LIN {X 123.176,Y 42.359,Z 55.000,A 180.000,B 0.000,C 180.000} C_DIS
LIN {X 122.928,Y 42.550,Z 55.000,A 180.000,B 0.000,C 180.000} C_DIS
LIN {X 122.818,Y 42.627,Z 55.000,A 180.000,B 0.000,C 180.000} C_DIS
LIN {X 122.639,Y 42.749,Z 55.000,A 180.000,B 0.000,C 180.000} C_DIS
LIN {X 122.461,Y 42.865,Z 55.000,A 180.000,B 0.000,C 180.000} C_DIS
LIN {X 122.282,Y 42.971,Z 55.000,A 180.000,B 0.000,C 180.000} C_DIS
LIN {X 122.103,Y 43.076,Z 55.000,A 180.000,B 0.000,C 180.000} C_DIS
LIN {X 121.731,Y 43.266,Z 55.000,A 180.000,B 0.000,C 180.000} C_DIS
LIN {X 121.567,Y 43.340,Z 55.000,A 180.000,B 0.000,C 180.000} C_DIS
LIN {X 121.325,Y 43.444,Z 55.000,A 180.000,B 0.000,C 180.000} C_DIS
LIN {X 121.209,Y 43.491,Z 55.000,A 180.000,B 0.000,C 180.000} C_DIS
LIN {X 120.841,Y 43.623,Z 55.000,A 180.000,B 0.000,C 180.000} C_DIS
LIN {X 120.673,Y 43.674,Z 55.000,A 180.000,B 0.000,C 180.000} C_DIS
LIN {X 120.494,Y 43.726,Z 55.000,A 180.000,B 0.000,C 180.000} C_DIS
LIN {X 120.315,Y 43.774,Z 55.000,A 180.000,B 0.000,C 180.000} C_DIS
LIN {X 119.958,Y 43.854,Z 55.000,A 180.000,B 0.000,C 180.000} C_DIS
LIN {X 119.779,Y 43.886,Z 55.000,A 180.000,B 0.000,C 180.000} C_DIS
LIN {X 119.632,Y 43.909,Z 55.000,A 180.000,B 0.000,C 180.000} C_DIS
; Link Move Starts
LIN {X 119.319,Y 43.951,Z 55.000,A 180.000,B 0.000,C 180.000} C_DIS
LIN {X 119.006,Y 43.981,Z 54.999,A 180.000,B 0.000,C 180.000} C_DIS
LIN {X 118.691,Y 43.993,Z 54.998,A 180.000,B 0.000,C 180.000} C_DIS
LIN {X 118.376,Y 43.995,Z 54.996,A 180.000,B 0.000,C 180.000} C_DIS
LIN {X 118.061,Y 43.985,Z 54.994,A 180.000,B 0.000,C 180.000} C_DIS
LIN {X 117.748,Y 43.957,Z 54.991,A 180.000,B 0.000,C 180.000} C_DIS
LIN {X 117.435,Y 43.920,Z 54.988,A 180.000,B 0.000,C 180.000} C_DIS
LIN {X 117.124,Y 43.871,Z 54.985,A 180.000,B 0.000,C 180.000} C_DIS
LIN {X 116.816,Y 43.804,Z 54.981,A 180.000,B 0.000,C 180.000} C_DIS
LIN {X 116.510,Y 43.727,Z 54.977,A 180.000,B 0.000,C 180.000} C_DIS
LIN {X 116.208,Y 43.639,Z 54.972,A 180.000,B 0.000,C 180.000} C_DIS
LIN {X 116.059,Y 43.587,Z 54.969,A 180.000,B 0.000,C 180.000} C_DIS
LIN {X 115.911,Y 43.534,Z 54.967,A 180.000,B 0.000,C 180.000} C_DIS
LIN {X 115.763,Y 43.481,Z 54.964,A 180.000,B 0.000,C 180.000} C_DIS
LIN {X 115.618,Y 43.419,Z 54.961,A 180.000,B 0.000,C 180.000} C_DIS
LIN {X 115.473,Y 43.357,Z 54.959,A 180.000,B 0.000,C 180.000} C_DIS
LIN {X 115.329,Y 43.294,Z 54.956,A 180.000,B 0.000,C 180.000} C_DIS
LIN {X 115.188,Y 43.224,Z 54.952,A 180.000,B 0.000,C 180.000} C_DIS
LIN {X 115.047,Y 43.153,Z 54.949,A 180.000,B 0.000,C 180.000} C_DIS
LIN {X 114.907,Y 43.081,Z 54.946,A 180.000,B 0.000,C 180.000} C_DIS
LIN {X 114.771,Y 43.002,Z 54.943,A 180.000,B 0.000,C 180.000} C_DIS
LIN {X 114.635,Y 42.922,Z 54.939,A 180.000,B 0.000,C 180.000} C_DIS
LIN {X 114.500,Y 42.842,Z 54.936,A 180.000,B 0.000,C 180.000} C_DIS
LIN {X 114.369,Y 42.754,Z 54.932,A 180.000,B 0.000,C 180.000} C_DIS
LIN {X 114.238,Y 42.666,Z 54.928,A 180.000,B 0.000,C 180.000} C_DIS
LIN {X 114.108,Y 42.577,Z 54.925,A 180.000,B 0.000,C 180.000} C_DIS
LIN {X 113.983,Y 42.482,Z 54.921,A 180.000,B 0.000,C 180.000} C_DIS
LIN {X 113.858,Y 42.385,Z 54.917,A 180.000,B 0.000,C 180.000} C_DIS
LIN {X 113.734,Y 42.289,Z 54.913,A 180.000,B 0.000,C 180.000} C_DIS
LIN {X 113.615,Y 42.185,Z 54.909,A 180.000,B 0.000,C 180.000} C_DIS
LIN {X 113.497,Y 42.081,Z 54.905,A 180.000,B 0.000,C 180.000} C_DIS
LIN {X 113.379,Y 41.977,Z 54.900,A 180.000,B 0.000,C 180.000} C_DIS
LIN {X 113.267,Y 41.866,Z 54.896,A 180.000,B 0.000,C 180.000} C_DIS
LIN {X 113.155,Y 41.755,Z 54.892,A 180.000,B 0.000,C 180.000} C_DIS
LIN {X 113.044,Y 41.644,Z 54.887,A 180.000,B 0.000,C 180.000} C_DIS
LIN {X 112.939,Y 41.526,Z 54.883,A 180.000,B 0.000,C 180.000} C_DIS
LIN {X 112.835,Y 41.408,Z 54.878,A 180.000,B 0.000,C 180.000} C_DIS
LIN {X 112.731,Y 41.290,Z 54.873,A 180.000,B 0.000,C 180.000} C_DIS
LIN {X 112.634,Y 41.166,Z 54.869,A 180.000,B 0.000,C 180.000} C_DIS
LIN {X 112.537,Y 41.041,Z 54.864,A 180.000,B 0.000,C 180.000} C_DIS
LIN {X 112.441,Y 40.917,Z 54.859,A 180.000,B 0.000,C 180.000} C_DIS
LIN {X 112.351,Y 40.787,Z 54.854,A 180.000,B 0.000,C 180.000} C_DIS
LIN {X 112.307,Y 40.722,Z 54.851,A 180.000,B 0.000,C 180.000} C_DIS
LIN {X 112.263,Y 40.657,Z 54.849,A 180.000,B 0.000,C 180.000} C_DIS
LIN {X 112.219,Y 40.592,Z 54.846,A 180.000,B 0.000,C 180.000} C_DIS
LIN {X 112.174,Y 40.526,Z 54.844,A 180.000,B 0.000,C 180.000} C_DIS
LIN {X 112.134,Y 40.459,Z 54.841,A 180.000,B 0.000,C 180.000} C_DIS
LIN {X 112.094,Y 40.391,Z 54.839,A 180.000,B 0.000,C 180.000} C_DIS
LIN {X 112.053,Y 40.323,Z 54.836,A 180.000,B 0.000,C 180.000} C_DIS
LIN {X 111.973,Y 40.188,Z 54.831,A 180.000,B 0.000,C 180.000} C_DIS
LIN {X 111.933,Y 40.120,Z 54.828,A 180.000,B 0.000,C 180.000} C_DIS
LIN {X 111.897,Y 40.050,Z 54.825,A 180.000,B 0.000,C 180.000} C_DIS
LIN {X 111.825,Y 39.910,Z 54.820,A 180.000,B 0.000,C 180.000} C_DIS
LIN {X 111.754,Y 39.769,Z 54.815,A 180.000,B 0.000,C 180.000} C_DIS
LIN {X 111.718,Y 39.699,Z 54.812,A 180.000,B 0.000,C 180.000} C_DIS
LIN {X 111.687,Y 39.627,Z 54.809,A 180.000,B 0.000,C 180.000} C_DIS
LIN {X 111.655,Y 39.555,Z 54.806,A 180.000,B 0.000,C 180.000} C_DIS
LIN {X 111.593,Y 39.410,Z 54.801,A 180.000,B 0.000,C 180.000} C_DIS
LIN {X 111.530,Y 39.266,Z 54.795,A 180.000,B 0.000,C 180.000} C_DIS
LIN {X 111.503,Y 39.192,Z 54.793,A 180.000,B 0.000,C 180.000} C_DIS
LIN {X 111.450,Y 39.044,Z 54.787,A 180.000,B 0.000,C 180.000} C_DIS
LIN {X 111.423,Y 38.969,Z 54.785,A 180.000,B 0.000,C 180.000} C_DIS
LIN {X 111.370,Y 38.821,Z 54.779,A 180.000,B 0.000,C 180.000} C_DIS
LIN {X 111.347,Y 38.746,Z 54.776,A 180.000,B 0.000,C 180.000} C_DIS
LIN {X 111.326,Y 38.670,Z 54.774,A 180.000,B 0.000,C 180.000} C_DIS
LIN {X 111.282,Y 38.519,Z 54.768,A 180.000,B 0.000,C 180.000} C_DIS
LIN {X 111.238,Y 38.368,Z 54.763,A 180.000,B 0.000,C 180.000} C_DIS
LIN {X 111.220,Y 38.291,Z 54.760,A 180.000,B 0.000,C 180.000} C_DIS
LIN {X 111.186,Y 38.137,Z 54.754,A 180.000,B 0.000,C 180.000} C_DIS
LIN {X 111.169,Y 38.060,Z 54.752,A 180.000,B 0.000,C 180.000} C_DIS
LIN {X 111.134,Y 37.906,Z 54.746,A 180.000,B 0.000,C 180.000} C_DIS
LIN {X 111.122,Y 37.829,Z 54.743,A 180.000,B 0.000,C 180.000} C_DIS
LIN {X 111.110,Y 37.751,Z 54.741,A 180.000,B 0.000,C 180.000} C_DIS
LIN {X 111.085,Y 37.595,Z 54.735,A 180.000,B 0.000,C 180.000} C_DIS
LIN {X 111.060,Y 37.440,Z 54.730,A 180.000,B 0.000,C 180.000} C_DIS
LIN {X 111.046,Y 37.283,Z 54.724,A 180.000,B 0.000,C 180.000} C_DIS
LIN {X 111.023,Y 37.048,Z 54.716,A 180.000,B 0.000,C 180.000} C_DIS
LIN {X 111.016,Y 36.969,Z 54.713,A 180.000,B 0.000,C 180.000} C_DIS
LIN {X 111.004,Y 36.576,Z 54.699,A 180.000,B 0.000,C 180.000} C_DIS
LIN {X 111.001,Y 36.497,Z 54.697,A 180.000,B 0.000,C 180.000} C_DIS
LIN {X 111.006,Y 36.340,Z 54.691,A 180.000,B 0.000,C 180.000} C_DIS
LIN {X 111.014,Y 36.103,Z 54.683,A 180.000,B 0.000,C 180.000} C_DIS
LIN {X 111.016,Y 36.025,Z 54.680,A 180.000,B 0.000,C 180.000} C_DIS
LIN {X 111.054,Y 35.633,Z 54.666,A 180.000,B 0.000,C 180.000} C_DIS
LIN {X 111.061,Y 35.554,Z 54.664,A 180.000,B 0.000,C 180.000} C_DIS
LIN {X 111.098,Y 35.321,Z 54.655,A 180.000,B 0.000,C 180.000} C_DIS
LIN {X 111.123,Y 35.165,Z 54.650,A 180.000,B 0.000,C 180.000} C_DIS
LIN {X 111.136,Y 35.088,Z 54.647,A 180.000,B 0.000,C 180.000} C_DIS
LIN {X 111.222,Y 34.703,Z 54.633,A 180.000,B 0.000,C 180.000} C_DIS
LIN {X 111.239,Y 34.627,Z 54.631,A 180.000,B 0.000,C 180.000} C_DIS
LIN {X 111.305,Y 34.400,Z 54.622,A 180.000,B 0.000,C 180.000} C_DIS
LIN {X 111.349,Y 34.248,Z 54.617,A 180.000,B 0.000,C 180.000} C_DIS
LIN {X 111.372,Y 34.173,Z 54.614,A 180.000,B 0.000,C 180.000} C_DIS
LIN {X 111.505,Y 33.802,Z 54.600,A 180.000,B 0.000,C 180.000} C_DIS
LIN {X 111.533,Y 33.729,Z 54.598,A 180.000,B 0.000,C 180.000} C_DIS
LIN {X 111.626,Y 33.512,Z 54.589,A 180.000,B 0.000,C 180.000} C_DIS
LIN {X 111.689,Y 33.367,Z 54.584,A 180.000,B 0.000,C 180.000} C_DIS
LIN {X 111.721,Y 33.295,Z 54.581,A 180.000,B 0.000,C 180.000} C_DIS
LIN {X 111.900,Y 32.944,Z 54.567,A 180.000,B 0.000,C 180.000} C_DIS
LIN {X 111.936,Y 32.875,Z 54.565,A 180.000,B 0.000,C 180.000} C_DIS
LIN {X 112.137,Y 32.536,Z 54.551,A 180.000,B 0.000,C 180.000} C_DIS
LIN {X 112.178,Y 32.468,Z 54.548,A 180.000,B 0.000,C 180.000} C_DIS
LIN {X 112.399,Y 32.143,Z 54.534,A 180.000,B 0.000,C 180.000} C_DIS
LIN {X 112.444,Y 32.078,Z 54.532,A 180.000,B 0.000,C 180.000} C_DIS
LIN {X 112.686,Y 31.767,Z 54.518,A 180.000,B 0.000,C 180.000} C_DIS
LIN {X 112.735,Y 31.706,Z 54.515,A 180.000,B 0.000,C 180.000} C_DIS
LIN {X 112.995,Y 31.410,Z 54.501,A 180.000,B 0.000,C 180.000} C_DIS
LIN {X 113.048,Y 31.352,Z 54.499,A 180.000,B 0.000,C 180.000} C_DIS
LIN {X 113.327,Y 31.074,Z 54.485,A 180.000,B 0.000,C 180.000} C_DIS
LIN {X 113.383,Y 31.019,Z 54.482,A 180.000,B 0.000,C 180.000} C_DIS
LIN {X 113.679,Y 30.759,Z 54.468,A 180.000,B 0.000,C 180.000} C_DIS
LIN {X 113.739,Y 30.708,Z 54.466,A 180.000,B 0.000,C 180.000} C_DIS
LIN {X 114.050,Y 30.466,Z 54.452,A 180.000,B 0.000,C 180.000} C_DIS
LIN {X 114.113,Y 30.419,Z 54.449,A 180.000,B 0.000,C 180.000} C_DIS
LIN {X 114.439,Y 30.198,Z 54.435,A 180.000,B 0.000,C 180.000} C_DIS
LIN {X 114.505,Y 30.155,Z 54.433,A 180.000,B 0.000,C 180.000} C_DIS
LIN {X 114.844,Y 29.955,Z 54.419,A 180.000,B 0.000,C 180.000} C_DIS
LIN {X 114.913,Y 29.916,Z 54.416,A 180.000,B 0.000,C 180.000} C_DIS
LIN {X 115.263,Y 29.737,Z 54.402,A 180.000,B 0.000,C 180.000} C_DIS
LIN {X 115.334,Y 29.703,Z 54.400,A 180.000,B 0.000,C 180.000} C_DIS
LIN {X 115.551,Y 29.609,Z 54.391,A 180.000,B 0.000,C 180.000} C_DIS
LIN {X 115.696,Y 29.547,Z 54.386,A 180.000,B 0.000,C 180.000} C_DIS
LIN {X 115.769,Y 29.517,Z 54.383,A 180.000,B 0.000,C 180.000} C_DIS
LIN {X 116.139,Y 29.384,Z 54.369,A 180.000,B 0.000,C 180.000} C_DIS
LIN {X 116.214,Y 29.359,Z 54.367,A 180.000,B 0.000,C 180.000} C_DIS
LIN {X 116.441,Y 29.293,Z 54.358,A 180.000,B 0.000,C 180.000} C_DIS
LIN {X 116.592,Y 29.249,Z 54.353,A 180.000,B 0.000,C 180.000} C_DIS
LIN {X 116.668,Y 29.229,Z 54.350,A 180.000,B 0.000,C 180.000} C_DIS
LIN {X 117.053,Y 29.144,Z 54.336,A 180.000,B 0.000,C 180.000} C_DIS
LIN {X 117.130,Y 29.129,Z 54.334,A 180.000,B 0.000,C 180.000} C_DIS
LIN {X 117.285,Y 29.104,Z 54.328,A 180.000,B 0.000,C 180.000} C_DIS
LIN {X 117.519,Y 29.067,Z 54.320,A 180.000,B 0.000,C 180.000} C_DIS
LIN {X 117.597,Y 29.057,Z 54.317,A 180.000,B 0.000,C 180.000} C_DIS
LIN {X 117.989,Y 29.020,Z 54.303,A 180.000,B 0.000,C 180.000} C_DIS
LIN {X 118.068,Y 29.015,Z 54.301,A 180.000,B 0.000,C 180.000} C_DIS
LIN {X 118.225,Y 29.010,Z 54.295,A 180.000,B 0.000,C 180.000} C_DIS
LIN {X 118.461,Y 29.002,Z 54.287,A 180.000,B 0.000,C 180.000} C_DIS
LIN {X 118.540,Y 29.002,Z 54.284,A 180.000,B 0.000,C 180.000} C_DIS
LIN {X 118.776,Y 29.010,Z 54.276,A 180.000,B 0.000,C 180.000} C_DIS
LIN {X 118.933,Y 29.015,Z 54.270,A 180.000,B 0.000,C 180.000} C_DIS
LIN {X 119.012,Y 29.020,Z 54.268,A 180.000,B 0.000,C 180.000} C_DIS
LIN {X 119.169,Y 29.035,Z 54.262,A 180.000,B 0.000,C 180.000} C_DIS
LIN {X 119.404,Y 29.057,Z 54.254,A 180.000,B 0.000,C 180.000} C_DIS
LIN {X 119.482,Y 29.067,Z 54.251,A 180.000,B 0.000,C 180.000} C_DIS
LIN {X 119.716,Y 29.104,Z 54.243,A 180.000,B 0.000,C 180.000} C_DIS
LIN {X 119.871,Y 29.129,Z 54.237,A 180.000,B 0.000,C 180.000} C_DIS
LIN {X 119.948,Y 29.144,Z 54.235,A 180.000,B 0.000,C 180.000} C_DIS
LIN {X 120.102,Y 29.178,Z 54.229,A 180.000,B 0.000,C 180.000} C_DIS
LIN {X 120.333,Y 29.230,Z 54.221,A 180.000,B 0.000,C 180.000} C_DIS
LIN {X 120.409,Y 29.250,Z 54.218,A 180.000,B 0.000,C 180.000} C_DIS
LIN {X 120.636,Y 29.316,Z 54.210,A 180.000,B 0.000,C 180.000} C_DIS
LIN {X 120.787,Y 29.359,Z 54.204,A 180.000,B 0.000,C 180.000} C_DIS
LIN {X 120.862,Y 29.384,Z 54.202,A 180.000,B 0.000,C 180.000} C_DIS
LIN {X 121.010,Y 29.438,Z 54.196,A 180.000,B 0.000,C 180.000} C_DIS
LIN {X 121.158,Y 29.491,Z 54.191,A 180.000,B 0.000,C 180.000} C_DIS
LIN {X 121.232,Y 29.518,Z 54.188,A 180.000,B 0.000,C 180.000} C_DIS
LIN {X 121.305,Y 29.547,Z 54.185,A 180.000,B 0.000,C 180.000} C_DIS
LIN {X 121.450,Y 29.610,Z 54.180,A 180.000,B 0.000,C 180.000} C_DIS
LIN {X 121.594,Y 29.672,Z 54.174,A 180.000,B 0.000,C 180.000} C_DIS
LIN {X 121.667,Y 29.704,Z 54.172,A 180.000,B 0.000,C 180.000} C_DIS
LIN {X 121.738,Y 29.738,Z 54.169,A 180.000,B 0.000,C 180.000} C_DIS
LIN {X 121.878,Y 29.809,Z 54.164,A 180.000,B 0.000,C 180.000} C_DIS
LIN {X 121.948,Y 29.845,Z 54.161,A 180.000,B 0.000,C 180.000} C_DIS
LIN {X 122.018,Y 29.881,Z 54.159,A 180.000,B 0.000,C 180.000} C_DIS
LIN {X 122.088,Y 29.917,Z 54.156,A 180.000,B 0.000,C 180.000} C_DIS
LIN {X 122.157,Y 29.955,Z 54.154,A 180.000,B 0.000,C 180.000} C_DIS
LIN {X 122.225,Y 29.995,Z 54.151,A 180.000,B 0.000,C 180.000} C_DIS
LIN {X 122.293,Y 30.035,Z 54.149,A 180.000,B 0.000,C 180.000} C_DIS
LIN {X 122.428,Y 30.115,Z 54.144,A 180.000,B 0.000,C 180.000} C_DIS
LIN {X 122.562,Y 30.198,Z 54.139,A 180.000,B 0.000,C 180.000} C_DIS
LIN {X 122.692,Y 30.287,Z 54.134,A 180.000,B 0.000,C 180.000} C_DIS
LIN {X 122.823,Y 30.376,Z 54.129,A 180.000,B 0.000,C 180.000} C_DIS
LIN {X 122.951,Y 30.467,Z 54.124,A 180.000,B 0.000,C 180.000} C_DIS
LIN {X 123.075,Y 30.563,Z 54.120,A 180.000,B 0.000,C 180.000} C_DIS
LIN {X 123.200,Y 30.660,Z 54.115,A 180.000,B 0.000,C 180.000} C_DIS
LIN {X 123.322,Y 30.759,Z 54.111,A 180.000,B 0.000,C 180.000} C_DIS
LIN {X 123.440,Y 30.863,Z 54.106,A 180.000,B 0.000,C 180.000} C_DIS
LIN {X 123.558,Y 30.968,Z 54.102,A 180.000,B 0.000,C 180.000} C_DIS
LIN {X 123.674,Y 31.074,Z 54.097,A 180.000,B 0.000,C 180.000} C_DIS
LIN {X 123.785,Y 31.186,Z 54.093,A 180.000,B 0.000,C 180.000} C_DIS
LIN {X 123.897,Y 31.297,Z 54.089,A 180.000,B 0.000,C 180.000} C_DIS
LIN {X 124.006,Y 31.411,Z 54.085,A 180.000,B 0.000,C 180.000} C_DIS
LIN {X 124.110,Y 31.529,Z 54.081,A 180.000,B 0.000,C 180.000} C_DIS
LIN {X 124.214,Y 31.647,Z 54.077,A 180.000,B 0.000,C 180.000} C_DIS
LIN {X 124.315,Y 31.768,Z 54.073,A 180.000,B 0.000,C 180.000} C_DIS
LIN {X 124.412,Y 31.893,Z 54.070,A 180.000,B 0.000,C 180.000} C_DIS
LIN {X 124.508,Y 32.017,Z 54.066,A 180.000,B 0.000,C 180.000} C_DIS
LIN {X 124.602,Y 32.144,Z 54.062,A 180.000,B 0.000,C 180.000} C_DIS
LIN {X 124.690,Y 32.274,Z 54.059,A 180.000,B 0.000,C 180.000} C_DIS
LIN {X 124.779,Y 32.404,Z 54.056,A 180.000,B 0.000,C 180.000} C_DIS
LIN {X 124.864,Y 32.537,Z 54.052,A 180.000,B 0.000,C 180.000} C_DIS
LIN {X 124.944,Y 32.672,Z 54.049,A 180.000,B 0.000,C 180.000} C_DIS
LIN {X 125.024,Y 32.808,Z 54.046,A 180.000,B 0.000,C 180.000} C_DIS
LIN {X 125.101,Y 32.945,Z 54.043,A 180.000,B 0.000,C 180.000} C_DIS
LIN {X 125.172,Y 33.086,Z 54.040,A 180.000,B 0.000,C 180.000} C_DIS
LIN {X 125.244,Y 33.226,Z 54.037,A 180.000,B 0.000,C 180.000} C_DIS
LIN {X 125.312,Y 33.368,Z 54.034,A 180.000,B 0.000,C 180.000} C_DIS
LIN {X 125.374,Y 33.513,Z 54.032,A 180.000,B 0.000,C 180.000} C_DIS
LIN {X 125.437,Y 33.657,Z 54.029,A 180.000,B 0.000,C 180.000} C_DIS
LIN {X 125.495,Y 33.804,Z 54.027,A 180.000,B 0.000,C 180.000} C_DIS
LIN {X 125.602,Y 34.100,Z 54.022,A 180.000,B 0.000,C 180.000} C_DIS
LIN {X 125.695,Y 34.401,Z 54.018,A 180.000,B 0.000,C 180.000} C_DIS
LIN {X 125.779,Y 34.705,Z 54.014,A 180.000,B 0.000,C 180.000} C_DIS
LIN {X 125.847,Y 35.012,Z 54.011,A 180.000,B 0.000,C 180.000} C_DIS
LIN {X 125.902,Y 35.322,Z 54.008,A 180.000,B 0.000,C 180.000} C_DIS
LIN {X 125.947,Y 35.634,Z 54.005,A 180.000,B 0.000,C 180.000} C_DIS
LIN {X 125.976,Y 35.947,Z 54.003,A 180.000,B 0.000,C 180.000} C_DIS
LIN {X 125.991,Y 36.262,Z 54.002,A 180.000,B 0.000,C 180.000} C_DIS
LIN {X 125.996,Y 36.577,Z 54.001,A 180.000,B 0.000,C 180.000} C_DIS
LIN {X 125.986,Y 36.892,Z 54.000,A 180.000,B 0.000,C 180.000} C_DIS
LIN {X 125.970,Y 37.123,Z 54.000,A 180.000,B 0.000,C 180.000} C_DIS
; Cutting Move Starts
LIN {X 125.947,Y 37.366,Z 54.000,A 180.000,B 0.000,C 180.000} C_DIS
LIN {X 125.923,Y 37.545,Z 54.000,A 180.000,B 0.000,C 180.000} C_DIS
LIN {X 125.866,Y 37.902,Z 54.000,A 180.000,B 0.000,C 180.000} C_DIS
LIN {X 125.857,Y 37.944,Z 54.000,A 180.000,B 0.000,C 180.000} C_DIS
LIN {X 125.787,Y 38.260,Z 54.000,A 180.000,B 0.000,C 180.000} C_DIS
LIN {X 125.742,Y 38.439,Z 54.000,A 180.000,B 0.000,C 180.000} C_DIS
LIN {X 125.638,Y 38.796,Z 54.000,A 180.000,B 0.000,C 180.000} C_DIS
LIN {X 125.575,Y 38.975,Z 54.000,A 180.000,B 0.000,C 180.000} C_DIS
LIN {X 125.500,Y 39.184,Z 54.000,A 180.000,B 0.000,C 180.000} C_DIS
LIN {X 125.441,Y 39.333,Z 54.000,A 180.000,B 0.000,C 180.000} C_DIS
LIN {X 125.286,Y 39.690,Z 54.000,A 180.000,B 0.000,C 180.000} C_DIS
LIN {X 125.195,Y 39.869,Z 54.000,A 180.000,B 0.000,C 180.000} C_DIS
LIN {X 125.104,Y 40.048,Z 54.000,A 180.000,B 0.000,C 180.000} C_DIS
LIN {X 125.004,Y 40.226,Z 54.000,A 180.000,B 0.000,C 180.000} C_DIS
LIN {X 124.898,Y 40.405,Z 54.000,A 180.000,B 0.000,C 180.000} C_DIS
LIN {X 124.787,Y 40.584,Z 54.000,A 180.000,B 0.000,C 180.000} C_DIS
LIN {X 124.606,Y 40.850,Z 54.000,A 180.000,B 0.000,C 180.000} C_DIS
LIN {X 124.540,Y 40.942,Z 54.000,A 180.000,B 0.000,C 180.000} C_DIS
LIN {X 124.402,Y 41.120,Z 54.000,A 180.000,B 0.000,C 180.000} C_DIS
LIN {X 124.261,Y 41.299,Z 54.000,A 180.000,B 0.000,C 180.000} C_DIS
LIN {X 124.070,Y 41.516,Z 54.000,A 180.000,B 0.000,C 180.000} C_DIS
LIN {X 123.943,Y 41.657,Z 54.000,A 180.000,B 0.000,C 180.000} C_DIS
LIN {X 123.712,Y 41.888,Z 54.000,A 180.000,B 0.000,C 180.000} C_DIS
LIN {X 123.579,Y 42.014,Z 54.000,A 180.000,B 0.000,C 180.000} C_DIS
LIN {X 123.354,Y 42.212,Z 54.000,A 180.000,B 0.000,C 180.000} C_DIS
LIN {X 123.176,Y 42.359,Z 54.000,A 180.000,B 0.000,C 180.000} C_DIS
LIN {X 122.928,Y 42.550,Z 54.000,A 180.000,B 0.000,C 180.000} C_DIS
LIN {X 122.818,Y 42.627,Z 54.000,A 180.000,B 0.000,C 180.000} C_DIS
LIN {X 122.639,Y 42.749,Z 54.000,A 180.000,B 0.000,C 180.000} C_DIS
LIN {X 122.461,Y 42.865,Z 54.000,A 180.000,B 0.000,C 180.000} C_DIS
LIN {X 122.282,Y 42.971,Z 54.000,A 180.000,B 0.000,C 180.000} C_DIS
LIN {X 122.103,Y 43.076,Z 54.000,A 180.000,B 0.000,C 180.000} C_DIS
LIN {X 121.731,Y 43.266,Z 54.000,A 180.000,B 0.000,C 180.000} C_DIS
LIN {X 121.567,Y 43.340,Z 54.000,A 180.000,B 0.000,C 180.000} C_DIS
LIN {X 121.325,Y 43.444,Z 54.000,A 180.000,B 0.000,C 180.000} C_DIS
LIN {X 121.209,Y 43.491,Z 54.000,A 180.000,B 0.000,C 180.000} C_DIS
LIN {X 120.841,Y 43.623,Z 54.000,A 180.000,B 0.000,C 180.000} C_DIS
LIN {X 120.673,Y 43.674,Z 54.000,A 180.000,B 0.000,C 180.000} C_DIS
LIN {X 120.494,Y 43.726,Z 54.000,A 180.000,B 0.000,C 180.000} C_DIS
LIN {X 120.315,Y 43.774,Z 54.000,A 180.000,B 0.000,C 180.000} C_DIS
LIN {X 119.958,Y 43.854,Z 54.000,A 180.000,B 0.000,C 180.000} C_DIS
LIN {X 119.779,Y 43.886,Z 54.000,A 180.000,B 0.000,C 180.000} C_DIS
LIN {X 119.632,Y 43.909,Z 54.000,A 180.000,B 0.000,C 180.000} C_DIS
LIN {X 119.600,Y 43.914,Z 54.000,A 180.000,B 0.000,C 180.000} C_DIS
LIN {X 119.422,Y 43.941,Z 54.000,A 180.000,B 0.000,C 180.000} C_DIS
LIN {X 119.006,Y 43.981,Z 54.000,A 180.000,B 0.000,C 180.000} C_DIS
LIN {X 118.885,Y 43.987,Z 54.000,A 180.000,B 0.000,C 180.000} C_DIS
LIN {X 118.528,Y 43.998,Z 54.000,A 180.000,B 0.000,C 180.000} C_DIS
LIN {X 118.349,Y 43.994,Z 54.000,A 180.000,B 0.000,C 180.000} C_DIS
LIN {X 118.170,Y 43.988,Z 54.000,A 180.000,B 0.000,C 180.000} C_DIS
LIN {X 117.994,Y 43.981,Z 54.000,A 180.000,B 0.000,C 180.000} C_DIS
LIN {X 117.634,Y 43.947,Z 54.000,A 180.000,B 0.000,C 180.000} C_DIS
LIN {X 117.455,Y 43.923,Z 54.000,A 180.000,B 0.000,C 180.000} C_DIS
LIN {X 117.098,Y 43.866,Z 54.000,A 180.000,B 0.000,C 180.000} C_DIS
LIN {X 116.919,Y 43.827,Z 54.000,A 180.000,B 0.000,C 180.000} C_DIS
LIN {X 116.740,Y 43.787,Z 54.000,A 180.000,B 0.000,C 180.000} C_DIS
LIN {X 116.561,Y 43.742,Z 54.000,A 180.000,B 0.000,C 180.000} C_DIS
LIN {X 116.204,Y 43.638,Z 54.000,A 180.000,B 0.000,C 180.000} C_DIS
LIN {X 116.159,Y 43.623,Z 54.000,A 180.000,B 0.000,C 180.000} C_DIS
LIN {X 115.846,Y 43.511,Z 54.000,A 180.000,B 0.000,C 180.000} C_DIS
LIN {X 115.675,Y 43.444,Z 54.000,A 180.000,B 0.000,C 180.000} C_DIS
LIN {X 115.310,Y 43.286,Z 54.000,A 180.000,B 0.000,C 180.000} C_DIS
LIN {X 115.269,Y 43.266,Z 54.000,A 180.000,B 0.000,C 180.000} C_DIS
LIN {X 114.918,Y 43.087,Z 54.000,A 180.000,B 0.000,C 180.000} C_DIS
LIN {X 114.774,Y 43.004,Z 54.000,A 180.000,B 0.000,C 180.000} C_DIS
LIN {X 114.595,Y 42.898,Z 54.000,A 180.000,B 0.000,C 180.000} C_DIS
LIN {X 114.416,Y 42.787,Z 54.000,A 180.000,B 0.000,C 180.000} C_DIS
LIN {X 114.237,Y 42.665,Z 54.000,A 180.000,B 0.000,C 180.000} C_DIS
LIN {X 114.072,Y 42.550,Z 54.000,A 180.000,B 0.000,C 180.000} C_DIS
LIN {X 113.841,Y 42.372,Z 54.000,A 180.000,B 0.000,C 180.000} C_DIS
LIN {X 113.701,Y 42.261,Z 54.000,A 180.000,B 0.000,C 180.000} C_DIS
LIN {X 113.421,Y 42.014,Z 54.000,A 180.000,B 0.000,C 180.000} C_DIS
LIN {X 113.343,Y 41.943,Z 54.000,A 180.000,B 0.000,C 180.000} C_DIS
LIN {X 113.057,Y 41.657,Z 54.000,A 180.000,B 0.000,C 180.000} C_DIS
LIN {X 112.986,Y 41.579,Z 54.000,A 180.000,B 0.000,C 180.000} C_DIS
LIN {X 112.739,Y 41.299,Z 54.000,A 180.000,B 0.000,C 180.000} C_DIS
LIN {X 112.628,Y 41.159,Z 54.000,A 180.000,B 0.000,C 180.000} C_DIS
LIN {X 112.450,Y 40.928,Z 54.000,A 180.000,B 0.000,C 180.000} C_DIS
LIN {X 112.335,Y 40.763,Z 54.000,A 180.000,B 0.000,C 180.000} C_DIS
LIN {X 112.213,Y 40.584,Z 54.000,A 180.000,B 0.000,C 180.000} C_DIS
LIN {X 112.102,Y 40.405,Z 54.000,A 180.000,B 0.000,C 180.000} C_DIS
LIN {X 111.996,Y 40.226,Z 54.000,A 180.000,B 0.000,C 180.000} C_DIS
LIN {X 111.913,Y 40.082,Z 54.000,A 180.000,B 0.000,C 180.000} C_DIS
LIN {X 111.734,Y 39.731,Z 54.000,A 180.000,B 0.000,C 180.000} C_DIS
LIN {X 111.714,Y 39.690,Z 54.000,A 180.000,B 0.000,C 180.000} C_DIS
LIN {X 111.556,Y 39.325,Z 54.000,A 180.000,B 0.000,C 180.000} C_DIS
LIN {X 111.489,Y 39.154,Z 54.000,A 180.000,B 0.000,C 180.000} C_DIS
LIN {X 111.377,Y 38.841,Z 54.000,A 180.000,B 0.000,C 180.000} C_DIS
LIN {X 111.362,Y 38.796,Z 54.000,A 180.000,B 0.000,C 180.000} C_DIS
LIN {X 111.258,Y 38.439,Z 54.000,A 180.000,B 0.000,C 180.000} C_DIS
LIN {X 111.213,Y 38.260,Z 54.000,A 180.000,B 0.000,C 180.000} C_DIS
LIN {X 111.173,Y 38.081,Z 54.000,A 180.000,B 0.000,C 180.000} C_DIS
LIN {X 111.134,Y 37.902,Z 54.000,A 180.000,B 0.000,C 180.000} C_DIS
LIN {X 111.077,Y 37.545,Z 54.000,A 180.000,B 0.000,C 180.000} C_DIS
LIN {X 111.053,Y 37.366,Z 54.000,A 180.000,B 0.000,C 180.000} C_DIS
LIN {X 111.019,Y 37.006,Z 54.000,A 180.000,B 0.000,C 180.000} C_DIS
LIN {X 111.012,Y 36.830,Z 54.000,A 180.000,B 0.000,C 180.000} C_DIS
LIN {X 111.006,Y 36.651,Z 54.000,A 180.000,B 0.000,C 180.000} C_DIS
LIN {X 111.002,Y 36.472,Z 54.000,A 180.000,B 0.000,C 180.000} C_DIS
LIN {X 111.013,Y 36.115,Z 54.000,A 180.000,B 0.000,C 180.000} C_DIS
LIN {X 111.019,Y 35.994,Z 54.000,A 180.000,B 0.000,C 180.000} C_DIS
LIN {X 111.059,Y 35.578,Z 54.000,A 180.000,B 0.000,C 180.000} C_DIS
LIN {X 111.086,Y 35.400,Z 54.000,A 180.000,B 0.000,C 180.000} C_DIS
LIN {X 111.114,Y 35.221,Z 54.000,A 180.000,B 0.000,C 180.000} C_DIS
LIN {X 111.146,Y 35.042,Z 54.000,A 180.000,B 0.000,C 180.000} C_DIS
LIN {X 111.226,Y 34.685,Z 54.000,A 180.000,B 0.000,C 180.000} C_DIS
LIN {X 111.274,Y 34.506,Z 54.000,A 180.000,B 0.000,C 180.000} C_DIS
LIN {X 111.326,Y 34.327,Z 54.000,A 180.000,B 0.000,C 180.000} C_DIS
LIN {X 111.377,Y 34.159,Z 54.000,A 180.000,B 0.000,C 180.000} C_DIS
LIN {X 111.509,Y 33.791,Z 54.000,A 180.000,B 0.000,C 180.000} C_DIS
LIN {X 111.556,Y 33.675,Z 54.000,A 180.000,B 0.000,C 180.000} C_DIS
LIN {X 111.660,Y 33.433,Z 54.000,A 180.000,B 0.000,C 180.000} C_DIS
LIN {X 111.734,Y 33.269,Z 54.000,A 180.000,B 0.000,C 180.000} C_DIS
LIN {X 111.924,Y 32.897,Z 54.000,A 180.000,B 0.000,C 180.000} C_DIS
LIN {X 112.029,Y 32.718,Z 54.000,A 180.000,B 0.000,C 180.000} C_DIS
LIN {X 112.135,Y 32.539,Z 54.000,A 180.000,B 0.000,C 180.000} C_DIS
LIN {X 112.251,Y 32.361,Z 54.000,A 180.000,B 0.000,C 180.000} C_DIS
LIN {X 112.373,Y 32.182,Z 54.000,A 180.000,B 0.000,C 180.000} C_DIS
LIN {X 112.450,Y 32.072,Z 54.000,A 180.000,B 0.000,C 180.000} C_DIS
LIN {X 112.641,Y 31.824,Z 54.000,A 180.000,B 0.000,C 180.000} C_DIS
LIN {X 112.788,Y 31.646,Z 54.000,A 180.000,B 0.000,C 180.000} C_DIS
LIN {X 112.986,Y 31.421,Z 54.000,A 180.000,B 0.000,C 180.000} C_DIS
LIN {X 113.112,Y 31.288,Z 54.000,A 180.000,B 0.000,C 180.000} C_DIS
LIN {X 113.343,Y 31.057,Z 54.000,A 180.000,B 0.000,C 180.000} C_DIS
LIN {X 113.484,Y 30.930,Z 54.000,A 180.000,B 0.000,C 180.000} C_DIS
LIN {X 113.701,Y 30.739,Z 54.000,A 180.000,B 0.000,C 180.000} C_DIS
LIN {X 113.880,Y 30.598,Z 54.000,A 180.000,B 0.000,C 180.000} C_DIS
LIN {X 114.058,Y 30.460,Z 54.000,A 180.000,B 0.000,C 180.000} C_DIS
LIN {X 114.150,Y 30.394,Z 54.000,A 180.000,B 0.000,C 180.000} C_DIS
LIN {X 114.416,Y 30.213,Z 54.000,A 180.000,B 0.000,C 180.000} C_DIS
LIN {X 114.595,Y 30.102,Z 54.000,A 180.000,B 0.000,C 180.000} C_DIS
LIN {X 114.774,Y 29.996,Z 54.000,A 180.000,B 0.000,C 180.000} C_DIS
LIN {X 114.952,Y 29.896,Z 54.000,A 180.000,B 0.000,C 180.000} C_DIS
LIN {X 115.131,Y 29.805,Z 54.000,A 180.000,B 0.000,C 180.000} C_DIS
LIN {X 115.310,Y 29.714,Z 54.000,A 180.000,B 0.000,C 180.000} C_DIS
LIN {X 115.667,Y 29.559,Z 54.000,A 180.000,B 0.000,C 180.000} C_DIS
LIN {X 115.816,Y 29.500,Z 54.000,A 180.000,B 0.000,C 180.000} C_DIS
LIN {X 116.025,Y 29.425,Z 54.000,A 180.000,B 0.000,C 180.000} C_DIS
LIN {X 116.204,Y 29.362,Z 54.000,A 180.000,B 0.000,C 180.000} C_DIS
LIN {X 116.561,Y 29.258,Z 54.000,A 180.000,B 0.000,C 180.000} C_DIS
LIN {X 116.740,Y 29.213,Z 54.000,A 180.000,B 0.000,C 180.000} C_DIS
LIN {X 117.056,Y 29.143,Z 54.000,A 180.000,B 0.000,C 180.000} C_DIS
LIN {X 117.098,Y 29.134,Z 54.000,A 180.000,B 0.000,C 180.000} C_DIS
LIN {X 117.455,Y 29.077,Z 54.000,A 180.000,B 0.000,C 180.000} C_DIS
LIN {X 117.634,Y 29.053,Z 54.000,A 180.000,B 0.000,C 180.000} C_DIS
LIN {X 117.991,Y 29.020,Z 54.000,A 180.000,B 0.000,C 180.000} C_DIS
LIN {X 118.170,Y 29.012,Z 54.000,A 180.000,B 0.000,C 180.000} C_DIS
LIN {X 118.349,Y 29.006,Z 54.000,A 180.000,B 0.000,C 180.000} C_DIS
LIN {X 118.528,Y 29.002,Z 54.000,A 180.000,B 0.000,C 180.000} C_DIS
LIN {X 118.885,Y 29.013,Z 54.000,A 180.000,B 0.000,C 180.000} C_DIS
LIN {X 119.064,Y 29.025,Z 54.000,A 180.000,B 0.000,C 180.000} C_DIS
LIN {X 119.422,Y 29.059,Z 54.000,A 180.000,B 0.000,C 180.000} C_DIS
LIN {X 119.600,Y 29.086,Z 54.000,A 180.000,B 0.000,C 180.000} C_DIS
LIN {X 119.779,Y 29.114,Z 54.000,A 180.000,B 0.000,C 180.000} C_DIS
LIN {X 119.944,Y 29.143,Z 54.000,A 180.000,B 0.000,C 180.000} C_DIS
LIN {X 120.315,Y 29.226,Z 54.000,A 180.000,B 0.000,C 180.000} C_DIS
LIN {X 120.494,Y 29.274,Z 54.000,A 180.000,B 0.000,C 180.000} C_DIS
LIN {X 120.673,Y 29.326,Z 54.000,A 180.000,B 0.000,C 180.000} C_DIS
LIN {X 120.852,Y 29.381,Z 54.000,A 180.000,B 0.000,C 180.000} C_DIS
LIN {X 121.209,Y 29.509,Z 54.000,A 180.000,B 0.000,C 180.000} C_DIS
LIN {X 121.388,Y 29.583,Z 54.000,A 180.000,B 0.000,C 180.000} C_DIS
LIN {X 121.610,Y 29.679,Z 54.000,A 180.000,B 0.000,C 180.000} C_DIS
LIN {X 121.746,Y 29.742,Z 54.000,A 180.000,B 0.000,C 180.000} C_DIS
LIN {X 122.103,Y 29.924,Z 54.000,A 180.000,B 0.000,C 180.000} C_DIS
LIN {X 122.282,Y 30.029,Z 54.000,A 180.000,B 0.000,C 180.000} C_DIS
LIN {X 122.461,Y 30.135,Z 54.000,A 180.000,B 0.000,C 180.000} C_DIS
LIN {X 122.587,Y 30.215,Z 54.000,A 180.000,B 0.000,C 180.000} C_DIS
LIN {X 122.850,Y 30.394,Z 54.000,A 180.000,B 0.000,C 180.000} C_DIS
LIN {X 122.997,Y 30.503,Z 54.000,A 180.000,B 0.000,C 180.000} C_DIS
LIN {X 123.176,Y 30.641,Z 54.000,A 180.000,B 0.000,C 180.000} C_DIS
LIN {X 123.313,Y 30.752,Z 54.000,A 180.000,B 0.000,C 180.000} C_DIS
LIN {X 123.533,Y 30.945,Z 54.000,A 180.000,B 0.000,C 180.000} C_DIS
LIN {X 123.709,Y 31.109,Z 54.000,A 180.000,B 0.000,C 180.000} C_DIS
LIN {X 123.891,Y 31.291,Z 54.000,A 180.000,B 0.000,C 180.000} C_DIS
LIN {X 124.055,Y 31.467,Z 54.000,A 180.000,B 0.000,C 180.000} C_DIS
LIN {X 124.248,Y 31.687,Z 54.000,A 180.000,B 0.000,C 180.000} C_DIS
LIN {X 124.359,Y 31.824,Z 54.000,A 180.000,B 0.000,C 180.000} C_DIS
LIN {X 124.497,Y 32.003,Z 54.000,A 180.000,B 0.000,C 180.000} C_DIS
LIN {X 124.606,Y 32.150,Z 54.000,A 180.000,B 0.000,C 180.000} C_DIS
LIN {X 124.785,Y 32.413,Z 54.000,A 180.000,B 0.000,C 180.000} C_DIS
LIN {X 124.865,Y 32.539,Z 54.000,A 180.000,B 0.000,C 180.000} C_DIS
LIN {X 124.971,Y 32.718,Z 54.000,A 180.000,B 0.000,C 180.000} C_DIS
LIN {X 125.076,Y 32.897,Z 54.000,A 180.000,B 0.000,C 180.000} C_DIS
LIN {X 125.258,Y 33.254,Z 54.000,A 180.000,B 0.000,C 180.000} C_DIS
LIN {X 125.321,Y 33.390,Z 54.000,A 180.000,B 0.000,C 180.000} C_DIS
LIN {X 125.417,Y 33.612,Z 54.000,A 180.000,B 0.000,C 180.000} C_DIS
LIN {X 125.491,Y 33.791,Z 54.000,A 180.000,B 0.000,C 180.000} C_DIS
LIN {X 125.619,Y 34.148,Z 54.000,A 180.000,B 0.000,C 180.000} C_DIS
LIN {X 125.674,Y 34.327,Z 54.000,A 180.000,B 0.000,C 180.000} C_DIS
LIN {X 125.726,Y 34.506,Z 54.000,A 180.000,B 0.000,C 180.000} C_DIS
LIN {X 125.774,Y 34.685,Z 54.000,A 180.000,B 0.000,C 180.000} C_DIS
LIN {X 125.857,Y 35.056,Z 54.000,A 180.000,B 0.000,C 180.000} C_DIS
LIN {X 125.886,Y 35.221,Z 54.000,A 180.000,B 0.000,C 180.000} C_DIS
LIN {X 125.914,Y 35.400,Z 54.000,A 180.000,B 0.000,C 180.000} C_DIS
LIN {X 125.941,Y 35.578,Z 54.000,A 180.000,B 0.000,C 180.000} C_DIS
LIN {X 125.975,Y 35.936,Z 54.000,A 180.000,B 0.000,C 180.000} C_DIS
LIN {X 125.987,Y 36.115,Z 54.000,A 180.000,B 0.000,C 180.000} C_DIS
LIN {X 125.998,Y 36.472,Z 54.000,A 180.000,B 0.000,C 180.000} C_DIS
LIN {X 125.994,Y 36.651,Z 54.000,A 180.000,B 0.000,C 180.000} C_DIS
LIN {X 125.988,Y 36.830,Z 54.000,A 180.000,B 0.000,C 180.000} C_DIS
LIN {X 125.980,Y 37.009,Z 54.000,A 180.000,B 0.000,C 180.000} C_DIS
LIN {X 125.970,Y 37.123,Z 54.000,A 180.000,B 0.000,C 180.000} C_DIS
; Link Move Starts
LIN {X 125.940,Y 37.437,Z 54.000,A 180.000,B 0.000,C 180.000} C_DIS
LIN {X 125.891,Y 37.748,Z 53.999,A 180.000,B 0.000,C 180.000} C_DIS
LIN {X 125.832,Y 38.057,Z 53.998,A 180.000,B 0.000,C 180.000} C_DIS
LIN {X 125.763,Y 38.365,Z 53.996,A 180.000,B 0.000,C 180.000} C_DIS
LIN {X 125.675,Y 38.667,Z 53.994,A 180.000,B 0.000,C 180.000} C_DIS
LIN {X 125.578,Y 38.967,Z 53.991,A 180.000,B 0.000,C 180.000} C_DIS
LIN {X 125.471,Y 39.263,Z 53.988,A 180.000,B 0.000,C 180.000} C_DIS
LIN {X 125.346,Y 39.552,Z 53.985,A 180.000,B 0.000,C 180.000} C_DIS
LIN {X 125.212,Y 39.837,Z 53.981,A 180.000,B 0.000,C 180.000} C_DIS
LIN {X 125.068,Y 40.118,Z 53.977,A 180.000,B 0.000,C 180.000} C_DIS
LIN {X 124.908,Y 40.389,Z 53.972,A 180.000,B 0.000,C 180.000} C_DIS
LIN {X 124.827,Y 40.524,Z 53.969,A 180.000,B 0.000,C 180.000} C_DIS
LIN {X 124.739,Y 40.654,Z 53.967,A 180.000,B 0.000,C 180.000} C_DIS
LIN {X 124.650,Y 40.785,Z 53.964,A 180.000,B 0.000,C 180.000} C_DIS
LIN {X 124.561,Y 40.915,Z 53.961,A 180.000,B 0.000,C 180.000} C_DIS
LIN {X 124.465,Y 41.039,Z 53.959,A 180.000,B 0.000,C 180.000} C_DIS
LIN {X 124.368,Y 41.164,Z 53.956,A 180.000,B 0.000,C 180.000} C_DIS
LIN {X 124.271,Y 41.288,Z 53.952,A 180.000,B 0.000,C 180.000} C_DIS
LIN {X 124.167,Y 41.406,Z 53.949,A 180.000,B 0.000,C 180.000} C_DIS
LIN {X 124.063,Y 41.524,Z 53.946,A 180.000,B 0.000,C 180.000} C_DIS
LIN {X 123.958,Y 41.642,Z 53.943,A 180.000,B 0.000,C 180.000} C_DIS
LIN {X 123.847,Y 41.753,Z 53.939,A 180.000,B 0.000,C 180.000} C_DIS
LIN {X 123.735,Y 41.864,Z 53.936,A 180.000,B 0.000,C 180.000} C_DIS
LIN {X 123.623,Y 41.975,Z 53.932,A 180.000,B 0.000,C 180.000} C_DIS
LIN {X 123.505,Y 42.079,Z 53.928,A 180.000,B 0.000,C 180.000} C_DIS
LIN {X 123.387,Y 42.183,Z 53.925,A 180.000,B 0.000,C 180.000} C_DIS
LIN {X 123.268,Y 42.287,Z 53.921,A 180.000,B 0.000,C 180.000} C_DIS
LIN {X 123.144,Y 42.383,Z 53.917,A 180.000,B 0.000,C 180.000} C_DIS
LIN {X 123.019,Y 42.480,Z 53.913,A 180.000,B 0.000,C 180.000} C_DIS
LIN {X 122.894,Y 42.576,Z 53.909,A 180.000,B 0.000,C 180.000} C_DIS
LIN {X 122.764,Y 42.664,Z 53.905,A 180.000,B 0.000,C 180.000} C_DIS
LIN {X 122.634,Y 42.753,Z 53.900,A 180.000,B 0.000,C 180.000} C_DIS
LIN {X 122.503,Y 42.840,Z 53.896,A 180.000,B 0.000,C 180.000} C_DIS
LIN {X 122.367,Y 42.921,Z 53.892,A 180.000,B 0.000,C 180.000} C_DIS
LIN {X 122.232,Y 43.001,Z 53.887,A 180.000,B 0.000,C 180.000} C_DIS
LIN {X 122.095,Y 43.080,Z 53.883,A 180.000,B 0.000,C 180.000} C_DIS
LIN {X 121.955,Y 43.151,Z 53.878,A 180.000,B 0.000,C 180.000} C_DIS
LIN {X 121.815,Y 43.223,Z 53.873,A 180.000,B 0.000,C 180.000} C_DIS
LIN {X 121.674,Y 43.293,Z 53.869,A 180.000,B 0.000,C 180.000} C_DIS
LIN {X 121.529,Y 43.356,Z 53.864,A 180.000,B 0.000,C 180.000} C_DIS
LIN {X 121.385,Y 43.418,Z 53.859,A 180.000,B 0.000,C 180.000} C_DIS
LIN {X 121.240,Y 43.480,Z 53.854,A 180.000,B 0.000,C 180.000} C_DIS
LIN {X 121.166,Y 43.506,Z 53.851,A 180.000,B 0.000,C 180.000} C_DIS
LIN {X 121.091,Y 43.533,Z 53.849,A 180.000,B 0.000,C 180.000} C_DIS
LIN {X 121.017,Y 43.560,Z 53.846,A 180.000,B 0.000,C 180.000} C_DIS
LIN {X 120.943,Y 43.586,Z 53.844,A 180.000,B 0.000,C 180.000} C_DIS
LIN {X 120.869,Y 43.613,Z 53.841,A 180.000,B 0.000,C 180.000} C_DIS
LIN {X 120.795,Y 43.638,Z 53.839,A 180.000,B 0.000,C 180.000} C_DIS
LIN {X 120.719,Y 43.660,Z 53.836,A 180.000,B 0.000,C 180.000} C_DIS
LIN {X 120.568,Y 43.704,Z 53.831,A 180.000,B 0.000,C 180.000} C_DIS
LIN {X 120.416,Y 43.748,Z 53.825,A 180.000,B 0.000,C 180.000} C_DIS
LIN {X 120.340,Y 43.769,Z 53.823,A 180.000,B 0.000,C 180.000} C_DIS
LIN {X 120.187,Y 43.803,Z 53.817,A 180.000,B 0.000,C 180.000} C_DIS
LIN {X 120.033,Y 43.837,Z 53.812,A 180.000,B 0.000,C 180.000} C_DIS
LIN {X 119.956,Y 43.855,Z 53.809,A 180.000,B 0.000,C 180.000} C_DIS
LIN {X 119.879,Y 43.870,Z 53.806,A 180.000,B 0.000,C 180.000} C_DIS
LIN {X 119.723,Y 43.895,Z 53.801,A 180.000,B 0.000,C 180.000} C_DIS
LIN {X 119.490,Y 43.932,Z 53.793,A 180.000,B 0.000,C 180.000} C_DIS
LIN {X 119.412,Y 43.942,Z 53.790,A 180.000,B 0.000,C 180.000} C_DIS
LIN {X 119.177,Y 43.965,Z 53.782,A 180.000,B 0.000,C 180.000} C_DIS
LIN {X 119.020,Y 43.979,Z 53.776,A 180.000,B 0.000,C 180.000} C_DIS
LIN {X 118.941,Y 43.985,Z 53.774,A 180.000,B 0.000,C 180.000} C_DIS
LIN {X 118.784,Y 43.990,Z 53.768,A 180.000,B 0.000,C 180.000} C_DIS
LIN {X 118.548,Y 43.997,Z 53.760,A 180.000,B 0.000,C 180.000} C_DIS
LIN {X 118.469,Y 43.998,Z 53.757,A 180.000,B 0.000,C 180.000} C_DIS
LIN {X 118.233,Y 43.990,Z 53.749,A 180.000,B 0.000,C 180.000} C_DIS
LIN {X 118.075,Y 43.985,Z 53.743,A 180.000,B 0.000,C 180.000} C_DIS
LIN {X 117.997,Y 43.981,Z 53.741,A 180.000,B 0.000,C 180.000} C_DIS
LIN {X 117.840,Y 43.966,Z 53.735,A 180.000,B 0.000,C 180.000} C_DIS
LIN {X 117.605,Y 43.944,Z 53.727,A 180.000,B 0.000,C 180.000} C_DIS
LIN {X 117.527,Y 43.934,Z 53.724,A 180.000,B 0.000,C 180.000} C_DIS
LIN {X 117.138,Y 43.873,Z 53.710,A 180.000,B 0.000,C 180.000} C_DIS
LIN {X 117.060,Y 43.858,Z 53.708,A 180.000,B 0.000,C 180.000} C_DIS
LIN {X 116.907,Y 43.824,Z 53.702,A 180.000,B 0.000,C 180.000} C_DIS
LIN {X 116.676,Y 43.772,Z 53.694,A 180.000,B 0.000,C 180.000} C_DIS
LIN {X 116.600,Y 43.753,Z 53.691,A 180.000,B 0.000,C 180.000} C_DIS
LIN {X 116.222,Y 43.643,Z 53.677,A 180.000,B 0.000,C 180.000} C_DIS
LIN {X 116.147,Y 43.619,Z 53.675,A 180.000,B 0.000,C 180.000} C_DIS
LIN {X 115.999,Y 43.565,Z 53.669,A 180.000,B 0.000,C 180.000} C_DIS
LIN {X 115.776,Y 43.485,Z 53.661,A 180.000,B 0.000,C 180.000} C_DIS
LIN {X 115.703,Y 43.456,Z 53.658,A 180.000,B 0.000,C 180.000} C_DIS
LIN {X 115.342,Y 43.300,Z 53.644,A 180.000,B 0.000,C 180.000} C_DIS
LIN {X 115.270,Y 43.266,Z 53.642,A 180.000,B 0.000,C 180.000} C_DIS
LIN {X 115.060,Y 43.159,Z 53.633,A 180.000,B 0.000,C 180.000} C_DIS
LIN {X 114.920,Y 43.088,Z 53.628,A 180.000,B 0.000,C 180.000} C_DIS
LIN {X 114.851,Y 43.049,Z 53.625,A 180.000,B 0.000,C 180.000} C_DIS
LIN {X 114.512,Y 42.849,Z 53.611,A 180.000,B 0.000,C 180.000} C_DIS
LIN {X 114.445,Y 42.807,Z 53.609,A 180.000,B 0.000,C 180.000} C_DIS
LIN {X 114.250,Y 42.674,Z 53.600,A 180.000,B 0.000,C 180.000} C_DIS
LIN {X 114.120,Y 42.585,Z 53.595,A 180.000,B 0.000,C 180.000} C_DIS
LIN {X 114.056,Y 42.539,Z 53.592,A 180.000,B 0.000,C 180.000} C_DIS
LIN {X 113.745,Y 42.297,Z 53.578,A 180.000,B 0.000,C 180.000} C_DIS
LIN {X 113.685,Y 42.247,Z 53.576,A 180.000,B 0.000,C 180.000} C_DIS
LIN {X 113.389,Y 41.986,Z 53.562,A 180.000,B 0.000,C 180.000} C_DIS
LIN {X 113.332,Y 41.932,Z 53.559,A 180.000,B 0.000,C 180.000} C_DIS
LIN {X 113.054,Y 41.654,Z 53.545,A 180.000,B 0.000,C 180.000} C_DIS
LIN {X 113.001,Y 41.596,Z 53.543,A 180.000,B 0.000,C 180.000} C_DIS
LIN {X 112.740,Y 41.300,Z 53.529,A 180.000,B 0.000,C 180.000} C_DIS
LIN {X 112.691,Y 41.239,Z 53.526,A 180.000,B 0.000,C 180.000} C_DIS
LIN {X 112.449,Y 40.928,Z 53.512,A 180.000,B 0.000,C 180.000} C_DIS
LIN {X 112.404,Y 40.864,Z 53.510,A 180.000,B 0.000,C 180.000} C_DIS
LIN {X 112.182,Y 40.538,Z 53.496,A 180.000,B 0.000,C 180.000} C_DIS
LIN {X 112.141,Y 40.471,Z 53.493,A 180.000,B 0.000,C 180.000} C_DIS
LIN {X 111.940,Y 40.132,Z 53.479,A 180.000,B 0.000,C 180.000} C_DIS
LIN {X 111.903,Y 40.063,Z 53.477,A 180.000,B 0.000,C 180.000} C_DIS
LIN {X 111.725,Y 39.712,Z 53.463,A 180.000,B 0.000,C 180.000} C_DIS
LIN {X 111.692,Y 39.640,Z 53.460,A 180.000,B 0.000,C 180.000} C_DIS
LIN {X 111.536,Y 39.279,Z 53.446,A 180.000,B 0.000,C 180.000} C_DIS
LIN {X 111.508,Y 39.205,Z 53.444,A 180.000,B 0.000,C 180.000} C_DIS
LIN {X 111.375,Y 38.835,Z 53.430,A 180.000,B 0.000,C 180.000} C_DIS
LIN {X 111.351,Y 38.759,Z 53.427,A 180.000,B 0.000,C 180.000} C_DIS
LIN {X 111.242,Y 38.381,Z 53.413,A 180.000,B 0.000,C 180.000} C_DIS
LIN {X 111.223,Y 38.305,Z 53.411,A 180.000,B 0.000,C 180.000} C_DIS
LIN {X 111.172,Y 38.074,Z 53.402,A 180.000,B 0.000,C 180.000} C_DIS
LIN {X 111.137,Y 37.920,Z 53.397,A 180.000,B 0.000,C 180.000} C_DIS
LIN {X 111.124,Y 37.843,Z 53.394,A 180.000,B 0.000,C 180.000} C_DIS
LIN {X 111.063,Y 37.454,Z 53.380,A 180.000,B 0.000,C 180.000} C_DIS
LIN {X 111.054,Y 37.375,Z 53.378,A 180.000,B 0.000,C 180.000} C_DIS
LIN {X 111.032,Y 37.140,Z 53.369,A 180.000,B 0.000,C 180.000} C_DIS
LIN {X 111.017,Y 36.983,Z 53.364,A 180.000,B 0.000,C 180.000} C_DIS
LIN {X 111.014,Y 36.905,Z 53.361,A 180.000,B 0.000,C 180.000} C_DIS
LIN {X 111.002,Y 36.511,Z 53.347,A 180.000,B 0.000,C 180.000} C_DIS
LIN {X 111.003,Y 36.432,Z 53.345,A 180.000,B 0.000,C 180.000} C_DIS
LIN {X 111.011,Y 36.196,Z 53.336,A 180.000,B 0.000,C 180.000} C_DIS
LIN {X 111.016,Y 36.039,Z 53.331,A 180.000,B 0.000,C 180.000} C_DIS
LIN {X 111.023,Y 35.960,Z 53.328,A 180.000,B 0.000,C 180.000} C_DIS
LIN {X 111.060,Y 35.568,Z 53.314,A 180.000,B 0.000,C 180.000} C_DIS
LIN {X 111.071,Y 35.490,Z 53.312,A 180.000,B 0.000,C 180.000} C_DIS
LIN {X 111.096,Y 35.335,Z 53.306,A 180.000,B 0.000,C 180.000} C_DIS
LIN {X 111.133,Y 35.102,Z 53.298,A 180.000,B 0.000,C 180.000} C_DIS
LIN {X 111.150,Y 35.025,Z 53.295,A 180.000,B 0.000,C 180.000} C_DIS
LIN {X 111.236,Y 34.640,Z 53.281,A 180.000,B 0.000,C 180.000} C_DIS
LIN {X 111.257,Y 34.565,Z 53.279,A 180.000,B 0.000,C 180.000} C_DIS
LIN {X 111.301,Y 34.413,Z 53.273,A 180.000,B 0.000,C 180.000} C_DIS
LIN {X 111.367,Y 34.186,Z 53.265,A 180.000,B 0.000,C 180.000} C_DIS
LIN {X 111.394,Y 34.112,Z 53.262,A 180.000,B 0.000,C 180.000} C_DIS
LIN {X 111.474,Y 33.890,Z 53.254,A 180.000,B 0.000,C 180.000} C_DIS
LIN {X 111.527,Y 33.742,Z 53.248,A 180.000,B 0.000,C 180.000} C_DIS
LIN {X 111.558,Y 33.669,Z 53.246,A 180.000,B 0.000,C 180.000} C_DIS
LIN {X 111.621,Y 33.525,Z 53.240,A 180.000,B 0.000,C 180.000} C_DIS
LIN {X 111.715,Y 33.308,Z 53.232,A 180.000,B 0.000,C 180.000} C_DIS
LIN {X 111.750,Y 33.238,Z 53.229,A 180.000,B 0.000,C 180.000} C_DIS
LIN {X 111.858,Y 33.027,Z 53.221,A 180.000,B 0.000,C 180.000} C_DIS
LIN {X 111.893,Y 32.957,Z 53.218,A 180.000,B 0.000,C 180.000} C_DIS
LIN {X 111.929,Y 32.887,Z 53.215,A 180.000,B 0.000,C 180.000} C_DIS
LIN {X 111.969,Y 32.819,Z 53.213,A 180.000,B 0.000,C 180.000} C_DIS
LIN {X 112.049,Y 32.684,Z 53.207,A 180.000,B 0.000,C 180.000} C_DIS
LIN {X 112.130,Y 32.548,Z 53.202,A 180.000,B 0.000,C 180.000} C_DIS
LIN {X 112.170,Y 32.480,Z 53.199,A 180.000,B 0.000,C 180.000} C_DIS
LIN {X 112.258,Y 32.350,Z 53.193,A 180.000,B 0.000,C 180.000} C_DIS
LIN {X 112.391,Y 32.155,Z 53.185,A 180.000,B 0.000,C 180.000} C_DIS
LIN {X 112.436,Y 32.090,Z 53.182,A 180.000,B 0.000,C 180.000} C_DIS
LIN {X 112.532,Y 31.965,Z 53.177,A 180.000,B 0.000,C 180.000} C_DIS
LIN {X 112.629,Y 31.841,Z 53.172,A 180.000,B 0.000,C 180.000} C_DIS
LIN {X 112.677,Y 31.778,Z 53.169,A 180.000,B 0.000,C 180.000} C_DIS
LIN {X 112.725,Y 31.716,Z 53.166,A 180.000,B 0.000,C 180.000} C_DIS
LIN {X 112.830,Y 31.598,Z 53.161,A 180.000,B 0.000,C 180.000} C_DIS
LIN {X 112.882,Y 31.539,Z 53.159,A 180.000,B 0.000,C 180.000} C_DIS
LIN {X 112.934,Y 31.480,Z 53.156,A 180.000,B 0.000,C 180.000} C_DIS
LIN {X 112.986,Y 31.421,Z 53.154,A 180.000,B 0.000,C 180.000} C_DIS
LIN {X 113.038,Y 31.362,Z 53.151,A 180.000,B 0.000,C 180.000} C_DIS
LIN {X 113.094,Y 31.306,Z 53.149,A 180.000,B 0.000,C 180.000} C_DIS
LIN {X 113.205,Y 31.195,Z 53.144,A 180.000,B 0.000,C 180.000} C_DIS
LIN {X 113.317,Y 31.084,Z 53.139,A 180.000,B 0.000,C 180.000} C_DIS
LIN {X 113.432,Y 30.976,Z 53.134,A 180.000,B 0.000,C 180.000} C_DIS
LIN {X 113.550,Y 30.872,Z 53.129,A 180.000,B 0.000,C 180.000} C_DIS
LIN {X 113.668,Y 30.768,Z 53.124,A 180.000,B 0.000,C 180.000} C_DIS
LIN {X 113.790,Y 30.668,Z 53.120,A 180.000,B 0.000,C 180.000} C_DIS
LIN {X 113.914,Y 30.571,Z 53.115,A 180.000,B 0.000,C 180.000} C_DIS
LIN {X 114.039,Y 30.475,Z 53.111,A 180.000,B 0.000,C 180.000} C_DIS
LIN {X 114.167,Y 30.383,Z 53.106,A 180.000,B 0.000,C 180.000} C_DIS
LIN {X 114.297,Y 30.294,Z 53.102,A 180.000,B 0.000,C 180.000} C_DIS
LIN {X 114.427,Y 30.206,Z 53.097,A 180.000,B 0.000,C 180.000} C_DIS
LIN {X 114.561,Y 30.122,Z 53.093,A 180.000,B 0.000,C 180.000} C_DIS
LIN {X 114.696,Y 30.042,Z 53.089,A 180.000,B 0.000,C 180.000} C_DIS
LIN {X 114.832,Y 29.962,Z 53.085,A 180.000,B 0.000,C 180.000} C_DIS
LIN {X 114.970,Y 29.887,Z 53.081,A 180.000,B 0.000,C 180.000} C_DIS
LIN {X 115.110,Y 29.815,Z 53.077,A 180.000,B 0.000,C 180.000} C_DIS
LIN {X 115.251,Y 29.744,Z 53.073,A 180.000,B 0.000,C 180.000} C_DIS
LIN {X 115.394,Y 29.678,Z 53.070,A 180.000,B 0.000,C 180.000} C_DIS
LIN {X 115.538,Y 29.615,Z 53.066,A 180.000,B 0.000,C 180.000} C_DIS
LIN {X 115.683,Y 29.552,Z 53.062,A 180.000,B 0.000,C 180.000} C_DIS
LIN {X 115.830,Y 29.495,Z 53.059,A 180.000,B 0.000,C 180.000} C_DIS
LIN {X 115.978,Y 29.442,Z 53.056,A 180.000,B 0.000,C 180.000} C_DIS
LIN {X 116.126,Y 29.389,Z 53.052,A 180.000,B 0.000,C 180.000} C_DIS
LIN {X 116.276,Y 29.341,Z 53.049,A 180.000,B 0.000,C 180.000} C_DIS
LIN {X 116.427,Y 29.297,Z 53.046,A 180.000,B 0.000,C 180.000} C_DIS
LIN {X 116.579,Y 29.253,Z 53.043,A 180.000,B 0.000,C 180.000} C_DIS
LIN {X 116.731,Y 29.215,Z 53.040,A 180.000,B 0.000,C 180.000} C_DIS
LIN {X 116.885,Y 29.181,Z 53.037,A 180.000,B 0.000,C 180.000} C_DIS
LIN {X 117.039,Y 29.147,Z 53.034,A 180.000,B 0.000,C 180.000} C_DIS
LIN {X 117.194,Y 29.118,Z 53.032,A 180.000,B 0.000,C 180.000} C_DIS
LIN {X 117.349,Y 29.094,Z 53.029,A 180.000,B 0.000,C 180.000} C_DIS
LIN {X 117.505,Y 29.069,Z 53.027,A 180.000,B 0.000,C 180.000} C_DIS
LIN {X 117.818,Y 29.036,Z 53.022,A 180.000,B 0.000,C 180.000} C_DIS
LIN {X 118.132,Y 29.013,Z 53.018,A 180.000,B 0.000,C 180.000} C_DIS
LIN {X 118.447,Y 29.003,Z 53.014,A 180.000,B 0.000,C 180.000} C_DIS
LIN {X 118.762,Y 29.009,Z 53.011,A 180.000,B 0.000,C 180.000} C_DIS
LIN {X 119.076,Y 29.026,Z 53.008,A 180.000,B 0.000,C 180.000} C_DIS
LIN {X 119.390,Y 29.056,Z 53.005,A 180.000,B 0.000,C 180.000} C_DIS
LIN {X 119.702,Y 29.102,Z 53.003,A 180.000,B 0.000,C 180.000} C_DIS
LIN {X 120.011,Y 29.158,Z 53.002,A 180.000,B 0.000,C 180.000} C_DIS
LIN {X 120.319,Y 29.227,Z 53.001,A 180.000,B 0.000,C 180.000} C_DIS
LIN {X 120.622,Y 29.312,Z 53.000,A 180.000,B 0.000,C 180.000} C_DIS
LIN {X 120.845,Y 29.379,Z 53.000,A 180.000,B 0.000,C 180.000} C_DIS
; Cutting Move Starts
LIN {X 120.852,Y 29.381,Z 53.000,A 180.000,B 0.000,C 180.000} C_DIS
LIN {X 121.209,Y 29.509,Z 53.000,A 180.000,B 0.000,C 180.000} C_DIS
LIN {X 121.388,Y 29.583,Z 53.000,A 180.000,B 0.000,C 180.000} C_DIS
LIN {X 121.610,Y 29.679,Z 53.000,A 180.000,B 0.000,C 180.000} C_DIS
LIN {X 121.746,Y 29.742,Z 53.000,A 180.000,B 0.000,C 180.000} C_DIS
LIN {X 122.103,Y 29.924,Z 53.000,A 180.000,B 0.000,C 180.000} C_DIS
LIN {X 122.282,Y 30.029,Z 53.000,A 180.000,B 0.000,C 180.000} C_DIS
LIN {X 122.461,Y 30.135,Z 53.000,A 180.000,B 0.000,C 180.000} C_DIS
LIN {X 122.587,Y 30.215,Z 53.000,A 180.000,B 0.000,C 180.000} C_DIS
LIN {X 122.850,Y 30.394,Z 53.000,A 180.000,B 0.000,C 180.000} C_DIS
LIN {X 122.997,Y 30.503,Z 53.000,A 180.000,B 0.000,C 180.000} C_DIS
LIN {X 123.176,Y 30.641,Z 53.000,A 180.000,B 0.000,C 180.000} C_DIS
LIN {X 123.313,Y 30.752,Z 53.000,A 180.000,B 0.000,C 180.000} C_DIS
LIN {X 123.533,Y 30.945,Z 53.000,A 180.000,B 0.000,C 180.000} C_DIS
LIN {X 123.709,Y 31.109,Z 53.000,A 180.000,B 0.000,C 180.000} C_DIS
LIN {X 123.891,Y 31.291,Z 53.000,A 180.000,B 0.000,C 180.000} C_DIS
LIN {X 124.055,Y 31.467,Z 53.000,A 180.000,B 0.000,C 180.000} C_DIS
LIN {X 124.248,Y 31.687,Z 53.000,A 180.000,B 0.000,C 180.000} C_DIS
LIN {X 124.359,Y 31.824,Z 53.000,A 180.000,B 0.000,C 180.000} C_DIS
LIN {X 124.497,Y 32.003,Z 53.000,A 180.000,B 0.000,C 180.000} C_DIS
LIN {X 124.606,Y 32.150,Z 53.000,A 180.000,B 0.000,C 180.000} C_DIS
LIN {X 124.785,Y 32.413,Z 53.000,A 180.000,B 0.000,C 180.000} C_DIS
LIN {X 124.865,Y 32.539,Z 53.000,A 180.000,B 0.000,C 180.000} C_DIS
LIN {X 124.971,Y 32.718,Z 53.000,A 180.000,B 0.000,C 180.000} C_DIS
LIN {X 125.076,Y 32.897,Z 53.000,A 180.000,B 0.000,C 180.000} C_DIS
LIN {X 125.258,Y 33.254,Z 53.000,A 180.000,B 0.000,C 180.000} C_DIS
LIN {X 125.321,Y 33.390,Z 53.000,A 180.000,B 0.000,C 180.000} C_DIS
LIN {X 125.417,Y 33.612,Z 53.000,A 180.000,B 0.000,C 180.000} C_DIS
LIN {X 125.491,Y 33.791,Z 53.000,A 180.000,B 0.000,C 180.000} C_DIS
LIN {X 125.619,Y 34.148,Z 53.000,A 180.000,B 0.000,C 180.000} C_DIS
LIN {X 125.674,Y 34.327,Z 53.000,A 180.000,B 0.000,C 180.000} C_DIS
LIN {X 125.726,Y 34.506,Z 53.000,A 180.000,B 0.000,C 180.000} C_DIS
LIN {X 125.774,Y 34.685,Z 53.000,A 180.000,B 0.000,C 180.000} C_DIS
LIN {X 125.857,Y 35.056,Z 53.000,A 180.000,B 0.000,C 180.000} C_DIS
LIN {X 125.886,Y 35.221,Z 53.000,A 180.000,B 0.000,C 180.000} C_DIS
LIN {X 125.914,Y 35.400,Z 53.000,A 180.000,B 0.000,C 180.000} C_DIS
LIN {X 125.941,Y 35.578,Z 53.000,A 180.000,B 0.000,C 180.000} C_DIS
LIN {X 125.975,Y 35.936,Z 53.000,A 180.000,B 0.000,C 180.000} C_DIS
LIN {X 125.987,Y 36.115,Z 53.000,A 180.000,B 0.000,C 180.000} C_DIS
LIN {X 125.998,Y 36.472,Z 53.000,A 180.000,B 0.000,C 180.000} C_DIS
LIN {X 125.994,Y 36.651,Z 53.000,A 180.000,B 0.000,C 180.000} C_DIS
LIN {X 125.988,Y 36.830,Z 53.000,A 180.000,B 0.000,C 180.000} C_DIS
LIN {X 125.980,Y 37.009,Z 53.000,A 180.000,B 0.000,C 180.000} C_DIS
LIN {X 125.947,Y 37.366,Z 53.000,A 180.000,B 0.000,C 180.000} C_DIS
LIN {X 125.923,Y 37.545,Z 53.000,A 180.000,B 0.000,C 180.000} C_DIS
LIN {X 125.866,Y 37.902,Z 53.000,A 180.000,B 0.000,C 180.000} C_DIS
LIN {X 125.857,Y 37.944,Z 53.000,A 180.000,B 0.000,C 180.000} C_DIS
LIN {X 125.787,Y 38.260,Z 53.000,A 180.000,B 0.000,C 180.000} C_DIS
LIN {X 125.742,Y 38.439,Z 53.000,A 180.000,B 0.000,C 180.000} C_DIS
LIN {X 125.638,Y 38.796,Z 53.000,A 180.000,B 0.000,C 180.000} C_DIS
LIN {X 125.575,Y 38.975,Z 53.000,A 180.000,B 0.000,C 180.000} C_DIS
LIN {X 125.500,Y 39.184,Z 53.000,A 180.000,B 0.000,C 180.000} C_DIS
LIN {X 125.441,Y 39.333,Z 53.000,A 180.000,B 0.000,C 180.000} C_DIS
LIN {X 125.286,Y 39.690,Z 53.000,A 180.000,B 0.000,C 180.000} C_DIS
LIN {X 125.195,Y 39.869,Z 53.000,A 180.000,B 0.000,C 180.000} C_DIS
LIN {X 125.104,Y 40.048,Z 53.000,A 180.000,B 0.000,C 180.000} C_DIS
LIN {X 125.004,Y 40.226,Z 53.000,A 180.000,B 0.000,C 180.000} C_DIS
LIN {X 124.898,Y 40.405,Z 53.000,A 180.000,B 0.000,C 180.000} C_DIS
LIN {X 124.787,Y 40.584,Z 53.000,A 180.000,B 0.000,C 180.000} C_DIS
LIN {X 124.606,Y 40.850,Z 53.000,A 180.000,B 0.000,C 180.000} C_DIS
LIN {X 124.540,Y 40.942,Z 53.000,A 180.000,B 0.000,C 180.000} C_DIS
LIN {X 124.402,Y 41.120,Z 53.000,A 180.000,B 0.000,C 180.000} C_DIS
LIN {X 124.261,Y 41.299,Z 53.000,A 180.000,B 0.000,C 180.000} C_DIS
LIN {X 124.070,Y 41.516,Z 53.000,A 180.000,B 0.000,C 180.000} C_DIS
LIN {X 123.943,Y 41.657,Z 53.000,A 180.000,B 0.000,C 180.000} C_DIS
LIN {X 123.712,Y 41.888,Z 53.000,A 180.000,B 0.000,C 180.000} C_DIS
LIN {X 123.579,Y 42.014,Z 53.000,A 180.000,B 0.000,C 180.000} C_DIS
LIN {X 123.354,Y 42.212,Z 53.000,A 180.000,B 0.000,C 180.000} C_DIS
LIN {X 123.176,Y 42.359,Z 53.000,A 180.000,B 0.000,C 180.000} C_DIS
LIN {X 122.928,Y 42.550,Z 53.000,A 180.000,B 0.000,C 180.000} C_DIS
LIN {X 122.818,Y 42.627,Z 53.000,A 180.000,B 0.000,C 180.000} C_DIS
LIN {X 122.639,Y 42.749,Z 53.000,A 180.000,B 0.000,C 180.000} C_DIS
LIN {X 122.461,Y 42.865,Z 53.000,A 180.000,B 0.000,C 180.000} C_DIS
LIN {X 122.282,Y 42.971,Z 53.000,A 180.000,B 0.000,C 180.000} C_DIS
LIN {X 122.103,Y 43.076,Z 53.000,A 180.000,B 0.000,C 180.000} C_DIS
LIN {X 121.731,Y 43.266,Z 53.000,A 180.000,B 0.000,C 180.000} C_DIS
LIN {X 121.567,Y 43.340,Z 53.000,A 180.000,B 0.000,C 180.000} C_DIS
LIN {X 121.325,Y 43.444,Z 53.000,A 180.000,B 0.000,C 180.000} C_DIS
LIN {X 121.209,Y 43.491,Z 53.000,A 180.000,B 0.000,C 180.000} C_DIS
LIN {X 120.841,Y 43.623,Z 53.000,A 180.000,B 0.000,C 180.000} C_DIS
LIN {X 120.673,Y 43.674,Z 53.000,A 180.000,B 0.000,C 180.000} C_DIS
LIN {X 120.494,Y 43.726,Z 53.000,A 180.000,B 0.000,C 180.000} C_DIS
LIN {X 120.315,Y 43.774,Z 53.000,A 180.000,B 0.000,C 180.000} C_DIS
LIN {X 119.958,Y 43.854,Z 53.000,A 180.000,B 0.000,C 180.000} C_DIS
LIN {X 119.779,Y 43.886,Z 53.000,A 180.000,B 0.000,C 180.000} C_DIS
LIN {X 119.600,Y 43.914,Z 53.000,A 180.000,B 0.000,C 180.000} C_DIS
LIN {X 119.422,Y 43.941,Z 53.000,A 180.000,B 0.000,C 180.000} C_DIS
LIN {X 119.006,Y 43.981,Z 53.000,A 180.000,B 0.000,C 180.000} C_DIS
LIN {X 118.885,Y 43.987,Z 53.000,A 180.000,B 0.000,C 180.000} C_DIS
LIN {X 118.528,Y 43.998,Z 53.000,A 180.000,B 0.000,C 180.000} C_DIS
LIN {X 118.349,Y 43.994,Z 53.000,A 180.000,B 0.000,C 180.000} C_DIS
LIN {X 118.170,Y 43.988,Z 53.000,A 180.000,B 0.000,C 180.000} C_DIS
LIN {X 117.994,Y 43.981,Z 53.000,A 180.000,B 0.000,C 180.000} C_DIS
LIN {X 117.634,Y 43.947,Z 53.000,A 180.000,B 0.000,C 180.000} C_DIS
LIN {X 117.455,Y 43.923,Z 53.000,A 180.000,B 0.000,C 180.000} C_DIS
LIN {X 117.098,Y 43.866,Z 53.000,A 180.000,B 0.000,C 180.000} C_DIS
LIN {X 116.919,Y 43.827,Z 53.000,A 180.000,B 0.000,C 180.000} C_DIS
LIN {X 116.740,Y 43.787,Z 53.000,A 180.000,B 0.000,C 180.000} C_DIS
LIN {X 116.561,Y 43.742,Z 53.000,A 180.000,B 0.000,C 180.000} C_DIS
LIN {X 116.204,Y 43.638,Z 53.000,A 180.000,B 0.000,C 180.000} C_DIS
LIN {X 116.159,Y 43.623,Z 53.000,A 180.000,B 0.000,C 180.000} C_DIS
LIN {X 115.846,Y 43.511,Z 53.000,A 180.000,B 0.000,C 180.000} C_DIS
LIN {X 115.675,Y 43.444,Z 53.000,A 180.000,B 0.000,C 180.000} C_DIS
LIN {X 115.310,Y 43.286,Z 53.000,A 180.000,B 0.000,C 180.000} C_DIS
LIN {X 115.269,Y 43.266,Z 53.000,A 180.000,B 0.000,C 180.000} C_DIS
LIN {X 114.918,Y 43.087,Z 53.000,A 180.000,B 0.000,C 180.000} C_DIS
LIN {X 114.774,Y 43.004,Z 53.000,A 180.000,B 0.000,C 180.000} C_DIS
LIN {X 114.595,Y 42.898,Z 53.000,A 180.000,B 0.000,C 180.000} C_DIS
LIN {X 114.416,Y 42.787,Z 53.000,A 180.000,B 0.000,C 180.000} C_DIS
LIN {X 114.237,Y 42.665,Z 53.000,A 180.000,B 0.000,C 180.000} C_DIS
LIN {X 114.072,Y 42.550,Z 53.000,A 180.000,B 0.000,C 180.000} C_DIS
LIN {X 113.841,Y 42.372,Z 53.000,A 180.000,B 0.000,C 180.000} C_DIS
LIN {X 113.701,Y 42.261,Z 53.000,A 180.000,B 0.000,C 180.000} C_DIS
LIN {X 113.421,Y 42.014,Z 53.000,A 180.000,B 0.000,C 180.000} C_DIS
LIN {X 113.343,Y 41.943,Z 53.000,A 180.000,B 0.000,C 180.000} C_DIS
LIN {X 113.057,Y 41.657,Z 53.000,A 180.000,B 0.000,C 180.000} C_DIS
LIN {X 112.986,Y 41.579,Z 53.000,A 180.000,B 0.000,C 180.000} C_DIS
LIN {X 112.739,Y 41.299,Z 53.000,A 180.000,B 0.000,C 180.000} C_DIS
LIN {X 112.628,Y 41.159,Z 53.000,A 180.000,B 0.000,C 180.000} C_DIS
LIN {X 112.450,Y 40.928,Z 53.000,A 180.000,B 0.000,C 180.000} C_DIS
LIN {X 112.335,Y 40.763,Z 53.000,A 180.000,B 0.000,C 180.000} C_DIS
LIN {X 112.213,Y 40.584,Z 53.000,A 180.000,B 0.000,C 180.000} C_DIS
LIN {X 112.102,Y 40.405,Z 53.000,A 180.000,B 0.000,C 180.000} C_DIS
LIN {X 111.996,Y 40.226,Z 53.000,A 180.000,B 0.000,C 180.000} C_DIS
LIN {X 111.913,Y 40.082,Z 53.000,A 180.000,B 0.000,C 180.000} C_DIS
LIN {X 111.734,Y 39.731,Z 53.000,A 180.000,B 0.000,C 180.000} C_DIS
LIN {X 111.714,Y 39.690,Z 53.000,A 180.000,B 0.000,C 180.000} C_DIS
LIN {X 111.556,Y 39.325,Z 53.000,A 180.000,B 0.000,C 180.000} C_DIS
LIN {X 111.489,Y 39.154,Z 53.000,A 180.000,B 0.000,C 180.000} C_DIS
LIN {X 111.377,Y 38.841,Z 53.000,A 180.000,B 0.000,C 180.000} C_DIS
LIN {X 111.362,Y 38.796,Z 53.000,A 180.000,B 0.000,C 180.000} C_DIS
LIN {X 111.258,Y 38.439,Z 53.000,A 180.000,B 0.000,C 180.000} C_DIS
LIN {X 111.213,Y 38.260,Z 53.000,A 180.000,B 0.000,C 180.000} C_DIS
LIN {X 111.173,Y 38.081,Z 53.000,A 180.000,B 0.000,C 180.000} C_DIS
LIN {X 111.134,Y 37.902,Z 53.000,A 180.000,B 0.000,C 180.000} C_DIS
LIN {X 111.077,Y 37.545,Z 53.000,A 180.000,B 0.000,C 180.000} C_DIS
LIN {X 111.053,Y 37.366,Z 53.000,A 180.000,B 0.000,C 180.000} C_DIS
LIN {X 111.019,Y 37.006,Z 53.000,A 180.000,B 0.000,C 180.000} C_DIS
LIN {X 111.012,Y 36.830,Z 53.000,A 180.000,B 0.000,C 180.000} C_DIS
LIN {X 111.006,Y 36.651,Z 53.000,A 180.000,B 0.000,C 180.000} C_DIS
LIN {X 111.002,Y 36.472,Z 53.000,A 180.000,B 0.000,C 180.000} C_DIS
LIN {X 111.013,Y 36.115,Z 53.000,A 180.000,B 0.000,C 180.000} C_DIS
LIN {X 111.019,Y 35.994,Z 53.000,A 180.000,B 0.000,C 180.000} C_DIS
LIN {X 111.059,Y 35.578,Z 53.000,A 180.000,B 0.000,C 180.000} C_DIS
LIN {X 111.086,Y 35.400,Z 53.000,A 180.000,B 0.000,C 180.000} C_DIS
LIN {X 111.114,Y 35.221,Z 53.000,A 180.000,B 0.000,C 180.000} C_DIS
LIN {X 111.146,Y 35.042,Z 53.000,A 180.000,B 0.000,C 180.000} C_DIS
LIN {X 111.226,Y 34.685,Z 53.000,A 180.000,B 0.000,C 180.000} C_DIS
LIN {X 111.274,Y 34.506,Z 53.000,A 180.000,B 0.000,C 180.000} C_DIS
LIN {X 111.326,Y 34.327,Z 53.000,A 180.000,B 0.000,C 180.000} C_DIS
LIN {X 111.377,Y 34.159,Z 53.000,A 180.000,B 0.000,C 180.000} C_DIS
LIN {X 111.509,Y 33.791,Z 53.000,A 180.000,B 0.000,C 180.000} C_DIS
LIN {X 111.556,Y 33.675,Z 53.000,A 180.000,B 0.000,C 180.000} C_DIS
LIN {X 111.660,Y 33.433,Z 53.000,A 180.000,B 0.000,C 180.000} C_DIS
LIN {X 111.734,Y 33.269,Z 53.000,A 180.000,B 0.000,C 180.000} C_DIS
LIN {X 111.924,Y 32.897,Z 53.000,A 180.000,B 0.000,C 180.000} C_DIS
LIN {X 112.029,Y 32.718,Z 53.000,A 180.000,B 0.000,C 180.000} C_DIS
LIN {X 112.135,Y 32.539,Z 53.000,A 180.000,B 0.000,C 180.000} C_DIS
LIN {X 112.251,Y 32.361,Z 53.000,A 180.000,B 0.000,C 180.000} C_DIS
LIN {X 112.373,Y 32.182,Z 53.000,A 180.000,B 0.000,C 180.000} C_DIS
LIN {X 112.450,Y 32.072,Z 53.000,A 180.000,B 0.000,C 180.000} C_DIS
LIN {X 112.641,Y 31.824,Z 53.000,A 180.000,B 0.000,C 180.000} C_DIS
LIN {X 112.788,Y 31.646,Z 53.000,A 180.000,B 0.000,C 180.000} C_DIS
LIN {X 112.986,Y 31.421,Z 53.000,A 180.000,B 0.000,C 180.000} C_DIS
LIN {X 113.112,Y 31.288,Z 53.000,A 180.000,B 0.000,C 180.000} C_DIS
LIN {X 113.343,Y 31.057,Z 53.000,A 180.000,B 0.000,C 180.000} C_DIS
LIN {X 113.484,Y 30.930,Z 53.000,A 180.000,B 0.000,C 180.000} C_DIS
LIN {X 113.701,Y 30.739,Z 53.000,A 180.000,B 0.000,C 180.000} C_DIS
LIN {X 113.880,Y 30.598,Z 53.000,A 180.000,B 0.000,C 180.000} C_DIS
LIN {X 114.058,Y 30.460,Z 53.000,A 180.000,B 0.000,C 180.000} C_DIS
LIN {X 114.150,Y 30.394,Z 53.000,A 180.000,B 0.000,C 180.000} C_DIS
LIN {X 114.416,Y 30.213,Z 53.000,A 180.000,B 0.000,C 180.000} C_DIS
LIN {X 114.595,Y 30.102,Z 53.000,A 180.000,B 0.000,C 180.000} C_DIS
LIN {X 114.774,Y 29.996,Z 53.000,A 180.000,B 0.000,C 180.000} C_DIS
LIN {X 114.952,Y 29.896,Z 53.000,A 180.000,B 0.000,C 180.000} C_DIS
LIN {X 115.131,Y 29.805,Z 53.000,A 180.000,B 0.000,C 180.000} C_DIS
LIN {X 115.310,Y 29.714,Z 53.000,A 180.000,B 0.000,C 180.000} C_DIS
LIN {X 115.667,Y 29.559,Z 53.000,A 180.000,B 0.000,C 180.000} C_DIS
LIN {X 115.816,Y 29.500,Z 53.000,A 180.000,B 0.000,C 180.000} C_DIS
LIN {X 116.025,Y 29.425,Z 53.000,A 180.000,B 0.000,C 180.000} C_DIS
LIN {X 116.204,Y 29.362,Z 53.000,A 180.000,B 0.000,C 180.000} C_DIS
LIN {X 116.561,Y 29.258,Z 53.000,A 180.000,B 0.000,C 180.000} C_DIS
LIN {X 116.740,Y 29.213,Z 53.000,A 180.000,B 0.000,C 180.000} C_DIS
LIN {X 117.056,Y 29.143,Z 53.000,A 180.000,B 0.000,C 180.000} C_DIS
LIN {X 117.098,Y 29.134,Z 53.000,A 180.000,B 0.000,C 180.000} C_DIS
LIN {X 117.455,Y 29.077,Z 53.000,A 180.000,B 0.000,C 180.000} C_DIS
LIN {X 117.634,Y 29.053,Z 53.000,A 180.000,B 0.000,C 180.000} C_DIS
LIN {X 117.991,Y 29.020,Z 53.000,A 180.000,B 0.000,C 180.000} C_DIS
LIN {X 118.170,Y 29.012,Z 53.000,A 180.000,B 0.000,C 180.000} C_DIS
LIN {X 118.349,Y 29.006,Z 53.000,A 180.000,B 0.000,C 180.000} C_DIS
LIN {X 118.528,Y 29.002,Z 53.000,A 180.000,B 0.000,C 180.000} C_DIS
LIN {X 118.885,Y 29.013,Z 53.000,A 180.000,B 0.000,C 180.000} C_DIS
LIN {X 119.064,Y 29.025,Z 53.000,A 180.000,B 0.000,C 180.000} C_DIS
LIN {X 119.422,Y 29.059,Z 53.000,A 180.000,B 0.000,C 180.000} C_DIS
LIN {X 119.600,Y 29.086,Z 53.000,A 180.000,B 0.000,C 180.000} C_DIS
LIN {X 119.779,Y 29.114,Z 53.000,A 180.000,B 0.000,C 180.000} C_DIS
LIN {X 119.944,Y 29.143,Z 53.000,A 180.000,B 0.000,C 180.000} C_DIS
LIN {X 120.315,Y 29.226,Z 53.000,A 180.000,B 0.000,C 180.000} C_DIS
LIN {X 120.494,Y 29.274,Z 53.000,A 180.000,B 0.000,C 180.000} C_DIS
LIN {X 120.673,Y 29.326,Z 53.000,A 180.000,B 0.000,C 180.000} C_DIS
LIN {X 120.845,Y 29.379,Z 53.000,A 180.000,B 0.000,C 180.000} C_DIS
; Link Move Starts
LIN {X 121.142,Y 29.485,Z 53.000,A 180.000,B 0.000,C 180.000} C_DIS
LIN {X 121.434,Y 29.603,Z 52.999,A 180.000,B 0.000,C 180.000} C_DIS
LIN {X 121.722,Y 29.730,Z 52.998,A 180.000,B 0.000,C 180.000} C_DIS
LIN {X 122.003,Y 29.873,Z 52.996,A 180.000,B 0.000,C 180.000} C_DIS
LIN {X 122.278,Y 30.026,Z 52.994,A 180.000,B 0.000,C 180.000} C_DIS
LIN {X 122.548,Y 30.189,Z 52.991,A 180.000,B 0.000,C 180.000} C_DIS
LIN {X 122.808,Y 30.366,Z 52.988,A 180.000,B 0.000,C 180.000} C_DIS
LIN {X 123.062,Y 30.553,Z 52.985,A 180.000,B 0.000,C 180.000} C_DIS
LIN {X 123.309,Y 30.748,Z 52.981,A 180.000,B 0.000,C 180.000} C_DIS
LIN {X 123.545,Y 30.956,Z 52.977,A 180.000,B 0.000,C 180.000} C_DIS
LIN {X 123.773,Y 31.174,Z 52.972,A 180.000,B 0.000,C 180.000} C_DIS
LIN {X 123.885,Y 31.285,Z 52.969,A 180.000,B 0.000,C 180.000} C_DIS
LIN {X 123.994,Y 31.398,Z 52.967,A 180.000,B 0.000,C 180.000} C_DIS
LIN {X 124.098,Y 31.516,Z 52.964,A 180.000,B 0.000,C 180.000} C_DIS
LIN {X 124.202,Y 31.634,Z 52.961,A 180.000,B 0.000,C 180.000} C_DIS
LIN {X 124.304,Y 31.754,Z 52.959,A 180.000,B 0.000,C 180.000} C_DIS
LIN {X 124.401,Y 31.879,Z 52.956,A 180.000,B 0.000,C 180.000} C_DIS
LIN {X 124.498,Y 32.003,Z 52.952,A 180.000,B 0.000,C 180.000} C_DIS
LIN {X 124.592,Y 32.129,Z 52.949,A 180.000,B 0.000,C 180.000} C_DIS
LIN {X 124.680,Y 32.260,Z 52.946,A 180.000,B 0.000,C 180.000} C_DIS
LIN {X 124.769,Y 32.390,Z 52.943,A 180.000,B 0.000,C 180.000} C_DIS
LIN {X 124.855,Y 32.522,Z 52.939,A 180.000,B 0.000,C 180.000} C_DIS
LIN {X 124.935,Y 32.657,Z 52.936,A 180.000,B 0.000,C 180.000} C_DIS
LIN {X 125.015,Y 32.793,Z 52.932,A 180.000,B 0.000,C 180.000} C_DIS
LIN {X 125.093,Y 32.930,Z 52.928,A 180.000,B 0.000,C 180.000} C_DIS
LIN {X 125.164,Y 33.070,Z 52.925,A 180.000,B 0.000,C 180.000} C_DIS
LIN {X 125.236,Y 33.211,Z 52.921,A 180.000,B 0.000,C 180.000} C_DIS
LIN {X 125.305,Y 33.352,Z 52.917,A 180.000,B 0.000,C 180.000} C_DIS
LIN {X 125.367,Y 33.497,Z 52.913,A 180.000,B 0.000,C 180.000} C_DIS
LIN {X 125.430,Y 33.641,Z 52.909,A 180.000,B 0.000,C 180.000} C_DIS
LIN {X 125.489,Y 33.787,Z 52.905,A 180.000,B 0.000,C 180.000} C_DIS
LIN {X 125.543,Y 33.935,Z 52.900,A 180.000,B 0.000,C 180.000} C_DIS
LIN {X 125.596,Y 34.084,Z 52.896,A 180.000,B 0.000,C 180.000} C_DIS
LIN {X 125.646,Y 34.233,Z 52.892,A 180.000,B 0.000,C 180.000} C_DIS
LIN {X 125.690,Y 34.384,Z 52.887,A 180.000,B 0.000,C 180.000} C_DIS
LIN {X 125.734,Y 34.535,Z 52.883,A 180.000,B 0.000,C 180.000} C_DIS
LIN {X 125.775,Y 34.688,Z 52.878,A 180.000,B 0.000,C 180.000} C_DIS
LIN {X 125.809,Y 34.841,Z 52.873,A 180.000,B 0.000,C 180.000} C_DIS
LIN {X 125.844,Y 34.995,Z 52.869,A 180.000,B 0.000,C 180.000} C_DIS
LIN {X 125.875,Y 35.149,Z 52.864,A 180.000,B 0.000,C 180.000} C_DIS
LIN {X 125.899,Y 35.305,Z 52.859,A 180.000,B 0.000,C 180.000} C_DIS
LIN {X 125.924,Y 35.460,Z 52.854,A 180.000,B 0.000,C 180.000} C_DIS
LIN {X 125.936,Y 35.538,Z 52.851,A 180.000,B 0.000,C 180.000} C_DIS
LIN {X 125.945,Y 35.617,Z 52.849,A 180.000,B 0.000,C 180.000} C_DIS
LIN {X 125.952,Y 35.695,Z 52.846,A 180.000,B 0.000,C 180.000} C_DIS
LIN {X 125.960,Y 35.773,Z 52.844,A 180.000,B 0.000,C 180.000} C_DIS
LIN {X 125.967,Y 35.852,Z 52.841,A 180.000,B 0.000,C 180.000} C_DIS
LIN {X 125.982,Y 36.009,Z 52.836,A 180.000,B 0.000,C 180.000} C_DIS
LIN {X 125.986,Y 36.087,Z 52.833,A 180.000,B 0.000,C 180.000} C_DIS
LIN {X 125.991,Y 36.245,Z 52.828,A 180.000,B 0.000,C 180.000} C_DIS
LIN {X 125.996,Y 36.402,Z 52.823,A 180.000,B 0.000,C 180.000} C_DIS
LIN {X 125.998,Y 36.481,Z 52.820,A 180.000,B 0.000,C 180.000} C_DIS
LIN {X 125.997,Y 36.560,Z 52.817,A 180.000,B 0.000,C 180.000} C_DIS
LIN {X 125.992,Y 36.717,Z 52.812,A 180.000,B 0.000,C 180.000} C_DIS
LIN {X 125.985,Y 36.953,Z 52.804,A 180.000,B 0.000,C 180.000} C_DIS
LIN {X 125.978,Y 37.032,Z 52.801,A 180.000,B 0.000,C 180.000} C_DIS
LIN {X 125.956,Y 37.267,Z 52.793,A 180.000,B 0.000,C 180.000} C_DIS
LIN {X 125.941,Y 37.424,Z 52.787,A 180.000,B 0.000,C 180.000} C_DIS
LIN {X 125.930,Y 37.502,Z 52.785,A 180.000,B 0.000,C 180.000} C_DIS
LIN {X 125.905,Y 37.657,Z 52.779,A 180.000,B 0.000,C 180.000} C_DIS
LIN {X 125.868,Y 37.891,Z 52.771,A 180.000,B 0.000,C 180.000} C_DIS
LIN {X 125.852,Y 37.968,Z 52.768,A 180.000,B 0.000,C 180.000} C_DIS
LIN {X 125.800,Y 38.198,Z 52.760,A 180.000,B 0.000,C 180.000} C_DIS
LIN {X 125.766,Y 38.352,Z 52.754,A 180.000,B 0.000,C 180.000} C_DIS
LIN {X 125.745,Y 38.428,Z 52.752,A 180.000,B 0.000,C 180.000} C_DIS
LIN {X 125.701,Y 38.579,Z 52.746,A 180.000,B 0.000,C 180.000} C_DIS
LIN {X 125.635,Y 38.806,Z 52.738,A 180.000,B 0.000,C 180.000} C_DIS
LIN {X 125.609,Y 38.880,Z 52.735,A 180.000,B 0.000,C 180.000} C_DIS
LIN {X 125.502,Y 39.177,Z 52.724,A 180.000,B 0.000,C 180.000} C_DIS
LIN {X 125.476,Y 39.251,Z 52.721,A 180.000,B 0.000,C 180.000} C_DIS
LIN {X 125.445,Y 39.323,Z 52.719,A 180.000,B 0.000,C 180.000} C_DIS
LIN {X 125.382,Y 39.468,Z 52.713,A 180.000,B 0.000,C 180.000} C_DIS
LIN {X 125.289,Y 39.685,Z 52.705,A 180.000,B 0.000,C 180.000} C_DIS
LIN {X 125.253,Y 39.755,Z 52.702,A 180.000,B 0.000,C 180.000} C_DIS
LIN {X 125.075,Y 40.106,Z 52.688,A 180.000,B 0.000,C 180.000} C_DIS
LIN {X 125.035,Y 40.174,Z 52.686,A 180.000,B 0.000,C 180.000} C_DIS
LIN {X 124.955,Y 40.310,Z 52.680,A 180.000,B 0.000,C 180.000} C_DIS
LIN {X 124.834,Y 40.513,Z 52.672,A 180.000,B 0.000,C 180.000} C_DIS
LIN {X 124.790,Y 40.578,Z 52.669,A 180.000,B 0.000,C 180.000} C_DIS
LIN {X 124.569,Y 40.904,Z 52.655,A 180.000,B 0.000,C 180.000} C_DIS
LIN {X 124.521,Y 40.966,Z 52.653,A 180.000,B 0.000,C 180.000} C_DIS
LIN {X 124.376,Y 41.153,Z 52.644,A 180.000,B 0.000,C 180.000} C_DIS
LIN {X 124.280,Y 41.278,Z 52.639,A 180.000,B 0.000,C 180.000} C_DIS
LIN {X 124.228,Y 41.337,Z 52.636,A 180.000,B 0.000,C 180.000} C_DIS
LIN {X 123.967,Y 41.632,Z 52.622,A 180.000,B 0.000,C 180.000} C_DIS
LIN {X 123.912,Y 41.688,Z 52.620,A 180.000,B 0.000,C 180.000} C_DIS
LIN {X 123.745,Y 41.855,Z 52.611,A 180.000,B 0.000,C 180.000} C_DIS
LIN {X 123.633,Y 41.966,Z 52.606,A 180.000,B 0.000,C 180.000} C_DIS
LIN {X 123.338,Y 42.227,Z 52.592,A 180.000,B 0.000,C 180.000} C_DIS
LIN {X 123.279,Y 42.279,Z 52.589,A 180.000,B 0.000,C 180.000} C_DIS
LIN {X 122.968,Y 42.520,Z 52.576,A 180.000,B 0.000,C 180.000} C_DIS
LIN {X 122.905,Y 42.568,Z 52.573,A 180.000,B 0.000,C 180.000} C_DIS
LIN {X 122.580,Y 42.790,Z 52.559,A 180.000,B 0.000,C 180.000} C_DIS
LIN {X 122.514,Y 42.834,Z 52.556,A 180.000,B 0.000,C 180.000} C_DIS
LIN {X 122.175,Y 43.034,Z 52.543,A 180.000,B 0.000,C 180.000} C_DIS
LIN {X 122.107,Y 43.074,Z 52.540,A 180.000,B 0.000,C 180.000} C_DIS
LIN {X 121.756,Y 43.253,Z 52.526,A 180.000,B 0.000,C 180.000} C_DIS
LIN {X 121.686,Y 43.288,Z 52.523,A 180.000,B 0.000,C 180.000} C_DIS
LIN {X 121.325,Y 43.444,Z 52.510,A 180.000,B 0.000,C 180.000} C_DIS
LIN {X 121.252,Y 43.475,Z 52.507,A 180.000,B 0.000,C 180.000} C_DIS
LIN {X 120.882,Y 43.609,Z 52.493,A 180.000,B 0.000,C 180.000} C_DIS
LIN {X 120.807,Y 43.635,Z 52.490,A 180.000,B 0.000,C 180.000} C_DIS
LIN {X 120.429,Y 43.744,Z 52.477,A 180.000,B 0.000,C 180.000} C_DIS
LIN {X 120.353,Y 43.766,Z 52.474,A 180.000,B 0.000,C 180.000} C_DIS
LIN {X 119.969,Y 43.852,Z 52.460,A 180.000,B 0.000,C 180.000} C_DIS
LIN {X 119.892,Y 43.868,Z 52.457,A 180.000,B 0.000,C 180.000} C_DIS
LIN {X 119.503,Y 43.930,Z 52.444,A 180.000,B 0.000,C 180.000} C_DIS
LIN {X 119.425,Y 43.941,Z 52.441,A 180.000,B 0.000,C 180.000} C_DIS
LIN {X 119.033,Y 43.978,Z 52.427,A 180.000,B 0.000,C 180.000} C_DIS
LIN {X 118.955,Y 43.984,Z 52.424,A 180.000,B 0.000,C 180.000} C_DIS
LIN {X 118.718,Y 43.992,Z 52.416,A 180.000,B 0.000,C 180.000} C_DIS
LIN {X 118.561,Y 43.997,Z 52.411,A 180.000,B 0.000,C 180.000} C_DIS
LIN {X 118.482,Y 43.998,Z 52.408,A 180.000,B 0.000,C 180.000} C_DIS
LIN {X 118.089,Y 43.986,Z 52.394,A 180.000,B 0.000,C 180.000} C_DIS
LIN {X 118.010,Y 43.982,Z 52.391,A 180.000,B 0.000,C 180.000} C_DIS
LIN {X 117.853,Y 43.967,Z 52.386,A 180.000,B 0.000,C 180.000} C_DIS
LIN {X 117.618,Y 43.945,Z 52.378,A 180.000,B 0.000,C 180.000} C_DIS
LIN {X 117.540,Y 43.936,Z 52.375,A 180.000,B 0.000,C 180.000} C_DIS
LIN {X 117.151,Y 43.875,Z 52.361,A 180.000,B 0.000,C 180.000} C_DIS
LIN {X 117.073,Y 43.861,Z 52.358,A 180.000,B 0.000,C 180.000} C_DIS
LIN {X 116.920,Y 43.827,Z 52.353,A 180.000,B 0.000,C 180.000} C_DIS
LIN {X 116.689,Y 43.775,Z 52.345,A 180.000,B 0.000,C 180.000} C_DIS
LIN {X 116.612,Y 43.757,Z 52.342,A 180.000,B 0.000,C 180.000} C_DIS
LIN {X 116.234,Y 43.647,Z 52.328,A 180.000,B 0.000,C 180.000} C_DIS
LIN {X 116.159,Y 43.623,Z 52.325,A 180.000,B 0.000,C 180.000} C_DIS
LIN {X 116.085,Y 43.597,Z 52.323,A 180.000,B 0.000,C 180.000} C_DIS
LIN {X 115.937,Y 43.543,Z 52.317,A 180.000,B 0.000,C 180.000} C_DIS
LIN {X 115.789,Y 43.490,Z 52.312,A 180.000,B 0.000,C 180.000} C_DIS
LIN {X 115.715,Y 43.462,Z 52.309,A 180.000,B 0.000,C 180.000} C_DIS
LIN {X 115.571,Y 43.399,Z 52.303,A 180.000,B 0.000,C 180.000} C_DIS
LIN {X 115.498,Y 43.368,Z 52.301,A 180.000,B 0.000,C 180.000} C_DIS
LIN {X 115.354,Y 43.305,Z 52.295,A 180.000,B 0.000,C 180.000} C_DIS
LIN {X 115.282,Y 43.272,Z 52.292,A 180.000,B 0.000,C 180.000} C_DIS
LIN {X 115.212,Y 43.237,Z 52.290,A 180.000,B 0.000,C 180.000} C_DIS
LIN {X 115.072,Y 43.165,Z 52.284,A 180.000,B 0.000,C 180.000} C_DIS
LIN {X 114.931,Y 43.094,Z 52.279,A 180.000,B 0.000,C 180.000} C_DIS
LIN {X 114.862,Y 43.056,Z 52.276,A 180.000,B 0.000,C 180.000} C_DIS
LIN {X 114.727,Y 42.976,Z 52.270,A 180.000,B 0.000,C 180.000} C_DIS
LIN {X 114.659,Y 42.936,Z 52.268,A 180.000,B 0.000,C 180.000} C_DIS
LIN {X 114.523,Y 42.856,Z 52.262,A 180.000,B 0.000,C 180.000} C_DIS
LIN {X 114.456,Y 42.814,Z 52.259,A 180.000,B 0.000,C 180.000} C_DIS
LIN {X 114.391,Y 42.770,Z 52.257,A 180.000,B 0.000,C 180.000} C_DIS
LIN {X 114.261,Y 42.681,Z 52.251,A 180.000,B 0.000,C 180.000} C_DIS
LIN {X 114.131,Y 42.593,Z 52.246,A 180.000,B 0.000,C 180.000} C_DIS
LIN {X 114.067,Y 42.547,Z 52.243,A 180.000,B 0.000,C 180.000} C_DIS
LIN {X 113.942,Y 42.450,Z 52.237,A 180.000,B 0.000,C 180.000} C_DIS
LIN {X 113.880,Y 42.402,Z 52.235,A 180.000,B 0.000,C 180.000} C_DIS
LIN {X 113.756,Y 42.305,Z 52.229,A 180.000,B 0.000,C 180.000} C_DIS
LIN {X 113.695,Y 42.256,Z 52.226,A 180.000,B 0.000,C 180.000} C_DIS
LIN {X 113.636,Y 42.203,Z 52.224,A 180.000,B 0.000,C 180.000} C_DIS
LIN {X 113.517,Y 42.099,Z 52.218,A 180.000,B 0.000,C 180.000} C_DIS
LIN {X 113.399,Y 41.995,Z 52.213,A 180.000,B 0.000,C 180.000} C_DIS
LIN {X 113.342,Y 41.941,Z 52.210,A 180.000,B 0.000,C 180.000} C_DIS
LIN {X 113.230,Y 41.830,Z 52.204,A 180.000,B 0.000,C 180.000} C_DIS
LIN {X 113.175,Y 41.774,Z 52.202,A 180.000,B 0.000,C 180.000} C_DIS
LIN {X 113.063,Y 41.663,Z 52.196,A 180.000,B 0.000,C 180.000} C_DIS
LIN {X 113.009,Y 41.606,Z 52.193,A 180.000,B 0.000,C 180.000} C_DIS
LIN {X 112.801,Y 41.369,Z 52.182,A 180.000,B 0.000,C 180.000} C_DIS
LIN {X 112.749,Y 41.310,Z 52.180,A 180.000,B 0.000,C 180.000} C_DIS
LIN {X 112.699,Y 41.250,Z 52.177,A 180.000,B 0.000,C 180.000} C_DIS
LIN {X 112.602,Y 41.125,Z 52.172,A 180.000,B 0.000,C 180.000} C_DIS
LIN {X 112.506,Y 41.001,Z 52.166,A 180.000,B 0.000,C 180.000} C_DIS
LIN {X 112.457,Y 40.939,Z 52.164,A 180.000,B 0.000,C 180.000} C_DIS
LIN {X 112.411,Y 40.875,Z 52.161,A 180.000,B 0.000,C 180.000} C_DIS
LIN {X 112.367,Y 40.810,Z 52.159,A 180.000,B 0.000,C 180.000} C_DIS
LIN {X 112.323,Y 40.745,Z 52.156,A 180.000,B 0.000,C 180.000} C_DIS
LIN {X 112.278,Y 40.679,Z 52.154,A 180.000,B 0.000,C 180.000} C_DIS
LIN {X 112.234,Y 40.614,Z 52.151,A 180.000,B 0.000,C 180.000} C_DIS
LIN {X 112.190,Y 40.549,Z 52.149,A 180.000,B 0.000,C 180.000} C_DIS
LIN {X 112.108,Y 40.415,Z 52.144,A 180.000,B 0.000,C 180.000} C_DIS
LIN {X 112.027,Y 40.279,Z 52.139,A 180.000,B 0.000,C 180.000} C_DIS
LIN {X 111.947,Y 40.144,Z 52.134,A 180.000,B 0.000,C 180.000} C_DIS
LIN {X 111.874,Y 40.004,Z 52.129,A 180.000,B 0.000,C 180.000} C_DIS
LIN {X 111.802,Y 39.864,Z 52.124,A 180.000,B 0.000,C 180.000} C_DIS
LIN {X 111.731,Y 39.724,Z 52.120,A 180.000,B 0.000,C 180.000} C_DIS
LIN {X 111.666,Y 39.580,Z 52.115,A 180.000,B 0.000,C 180.000} C_DIS
LIN {X 111.604,Y 39.436,Z 52.111,A 180.000,B 0.000,C 180.000} C_DIS
LIN {X 111.541,Y 39.291,Z 52.106,A 180.000,B 0.000,C 180.000} C_DIS
LIN {X 111.486,Y 39.143,Z 52.102,A 180.000,B 0.000,C 180.000} C_DIS
LIN {X 111.432,Y 38.995,Z 52.097,A 180.000,B 0.000,C 180.000} C_DIS
LIN {X 111.379,Y 38.847,Z 52.093,A 180.000,B 0.000,C 180.000} C_DIS
LIN {X 111.333,Y 38.696,Z 52.089,A 180.000,B 0.000,C 180.000} C_DIS
LIN {X 111.289,Y 38.545,Z 52.085,A 180.000,B 0.000,C 180.000} C_DIS
LIN {X 111.245,Y 38.394,Z 52.081,A 180.000,B 0.000,C 180.000} C_DIS
LIN {X 111.209,Y 38.241,Z 52.077,A 180.000,B 0.000,C 180.000} C_DIS
LIN {X 111.175,Y 38.087,Z 52.073,A 180.000,B 0.000,C 180.000} C_DIS
LIN {X 111.140,Y 37.933,Z 52.070,A 180.000,B 0.000,C 180.000} C_DIS
LIN {X 111.114,Y 37.778,Z 52.066,A 180.000,B 0.000,C 180.000} C_DIS
LIN {X 111.089,Y 37.622,Z 52.062,A 180.000,B 0.000,C 180.000} C_DIS
LIN {X 111.065,Y 37.467,Z 52.059,A 180.000,B 0.000,C 180.000} C_DIS
LIN {X 111.048,Y 37.310,Z 52.056,A 180.000,B 0.000,C 180.000} C_DIS
LIN {X 111.033,Y 37.153,Z 52.052,A 180.000,B 0.000,C 180.000} C_DIS
LIN {X 111.018,Y 36.997,Z 52.049,A 180.000,B 0.000,C 180.000} C_DIS
LIN {X 111.012,Y 36.839,Z 52.046,A 180.000,B 0.000,C 180.000} C_DIS
LIN {X 111.007,Y 36.682,Z 52.043,A 180.000,B 0.000,C 180.000} C_DIS
LIN {X 111.002,Y 36.524,Z 52.040,A 180.000,B 0.000,C 180.000} C_DIS
LIN {X 111.005,Y 36.367,Z 52.037,A 180.000,B 0.000,C 180.000} C_DIS
LIN {X 111.010,Y 36.210,Z 52.034,A 180.000,B 0.000,C 180.000} C_DIS
LIN {X 111.015,Y 36.052,Z 52.032,A 180.000,B 0.000,C 180.000} C_DIS
LIN {X 111.029,Y 35.895,Z 52.029,A 180.000,B 0.000,C 180.000} C_DIS
LIN {X 111.044,Y 35.738,Z 52.027,A 180.000,B 0.000,C 180.000} C_DIS
LIN {X 111.082,Y 35.426,Z 52.022,A 180.000,B 0.000,C 180.000} C_DIS
LIN {X 111.131,Y 35.115,Z 52.018,A 180.000,B 0.000,C 180.000} C_DIS
LIN {X 111.198,Y 34.807,Z 52.014,A 180.000,B 0.000,C 180.000} C_DIS
LIN {X 111.276,Y 34.502,Z 52.011,A 180.000,B 0.000,C 180.000} C_DIS
LIN {X 111.363,Y 34.199,Z 52.008,A 180.000,B 0.000,C 180.000} C_DIS
LIN {X 111.469,Y 33.902,Z 52.005,A 180.000,B 0.000,C 180.000} C_DIS
LIN {X 111.584,Y 33.609,Z 52.003,A 180.000,B 0.000,C 180.000} C_DIS
LIN {X 111.709,Y 33.320,Z 52.002,A 180.000,B 0.000,C 180.000} C_DIS
LIN {X 111.852,Y 33.039,Z 52.001,A 180.000,B 0.000,C 180.000} C_DIS
LIN {X 112.003,Y 32.763,Z 52.000,A 180.000,B 0.000,C 180.000} C_DIS
LIN {X 112.121,Y 32.562,Z 52.000,A 180.000,B 0.000,C 180.000} C_DIS
; Cutting Move Starts
LIN {X 112.135,Y 32.539,Z 52.000,A 180.000,B 0.000,C 180.000} C_DIS
LIN {X 112.251,Y 32.361,Z 52.000,A 180.000,B 0.000,C 180.000} C_DIS
LIN {X 112.373,Y 32.182,Z 52.000,A 180.000,B 0.000,C 180.000} C_DIS
LIN {X 112.450,Y 32.072,Z 52.000,A 180.000,B 0.000,C 180.000} C_DIS
LIN {X 112.641,Y 31.824,Z 52.000,A 180.000,B 0.000,C 180.000} C_DIS
LIN {X 112.788,Y 31.646,Z 52.000,A 180.000,B 0.000,C 180.000} C_DIS
LIN {X 112.986,Y 31.421,Z 52.000,A 180.000,B 0.000,C 180.000} C_DIS
LIN {X 113.112,Y 31.288,Z 52.000,A 180.000,B 0.000,C 180.000} C_DIS
LIN {X 113.343,Y 31.057,Z 52.000,A 180.000,B 0.000,C 180.000} C_DIS
LIN {X 113.484,Y 30.930,Z 52.000,A 180.000,B 0.000,C 180.000} C_DIS
LIN {X 113.701,Y 30.739,Z 52.000,A 180.000,B 0.000,C 180.000} C_DIS
LIN {X 113.880,Y 30.598,Z 52.000,A 180.000,B 0.000,C 180.000} C_DIS
LIN {X 114.058,Y 30.460,Z 52.000,A 180.000,B 0.000,C 180.000} C_DIS
LIN {X 114.150,Y 30.394,Z 52.000,A 180.000,B 0.000,C 180.000} C_DIS
LIN {X 114.416,Y 30.213,Z 52.000,A 180.000,B 0.000,C 180.000} C_DIS
LIN {X 114.595,Y 30.102,Z 52.000,A 180.000,B 0.000,C 180.000} C_DIS
LIN {X 114.774,Y 29.996,Z 52.000,A 180.000,B 0.000,C 180.000} C_DIS
LIN {X 114.952,Y 29.896,Z 52.000,A 180.000,B 0.000,C 180.000} C_DIS
LIN {X 115.131,Y 29.805,Z 52.000,A 180.000,B 0.000,C 180.000} C_DIS
LIN {X 115.310,Y 29.714,Z 52.000,A 180.000,B 0.000,C 180.000} C_DIS
LIN {X 115.667,Y 29.559,Z 52.000,A 180.000,B 0.000,C 180.000} C_DIS
LIN {X 115.816,Y 29.500,Z 52.000,A 180.000,B 0.000,C 180.000} C_DIS
LIN {X 116.025,Y 29.425,Z 52.000,A 180.000,B 0.000,C 180.000} C_DIS
LIN {X 116.204,Y 29.362,Z 52.000,A 180.000,B 0.000,C 180.000} C_DIS
LIN {X 116.561,Y 29.258,Z 52.000,A 180.000,B 0.000,C 180.000} C_DIS
LIN {X 116.740,Y 29.213,Z 52.000,A 180.000,B 0.000,C 180.000} C_DIS
LIN {X 117.056,Y 29.143,Z 52.000,A 180.000,B 0.000,C 180.000} C_DIS
LIN {X 117.098,Y 29.134,Z 52.000,A 180.000,B 0.000,C 180.000} C_DIS
LIN {X 117.455,Y 29.077,Z 52.000,A 180.000,B 0.000,C 180.000} C_DIS
LIN {X 117.634,Y 29.053,Z 52.000,A 180.000,B 0.000,C 180.000} C_DIS
LIN {X 117.991,Y 29.020,Z 52.000,A 180.000,B 0.000,C 180.000} C_DIS
LIN {X 118.170,Y 29.012,Z 52.000,A 180.000,B 0.000,C 180.000} C_DIS
LIN {X 118.349,Y 29.006,Z 52.000,A 180.000,B 0.000,C 180.000} C_DIS
LIN {X 118.528,Y 29.002,Z 52.000,A 180.000,B 0.000,C 180.000} C_DIS
LIN {X 118.885,Y 29.013,Z 52.000,A 180.000,B 0.000,C 180.000} C_DIS
LIN {X 119.064,Y 29.025,Z 52.000,A 180.000,B 0.000,C 180.000} C_DIS
LIN {X 119.422,Y 29.059,Z 52.000,A 180.000,B 0.000,C 180.000} C_DIS
LIN {X 119.600,Y 29.086,Z 52.000,A 180.000,B 0.000,C 180.000} C_DIS
LIN {X 119.779,Y 29.114,Z 52.000,A 180.000,B 0.000,C 180.000} C_DIS
LIN {X 119.944,Y 29.143,Z 52.000,A 180.000,B 0.000,C 180.000} C_DIS
LIN {X 120.315,Y 29.226,Z 52.000,A 180.000,B 0.000,C 180.000} C_DIS
LIN {X 120.494,Y 29.274,Z 52.000,A 180.000,B 0.000,C 180.000} C_DIS
LIN {X 120.673,Y 29.326,Z 52.000,A 180.000,B 0.000,C 180.000} C_DIS
LIN {X 120.845,Y 29.379,Z 52.000,A 180.000,B 0.000,C 180.000} C_DIS
LIN {X 120.852,Y 29.381,Z 52.000,A 180.000,B 0.000,C 180.000} C_DIS
LIN {X 121.209,Y 29.509,Z 52.000,A 180.000,B 0.000,C 180.000} C_DIS
LIN {X 121.388,Y 29.583,Z 52.000,A 180.000,B 0.000,C 180.000} C_DIS
LIN {X 121.610,Y 29.679,Z 52.000,A 180.000,B 0.000,C 180.000} C_DIS
LIN {X 121.746,Y 29.742,Z 52.000,A 180.000,B 0.000,C 180.000} C_DIS
LIN {X 122.103,Y 29.924,Z 52.000,A 180.000,B 0.000,C 180.000} C_DIS
LIN {X 122.282,Y 30.029,Z 52.000,A 180.000,B 0.000,C 180.000} C_DIS
LIN {X 122.461,Y 30.135,Z 52.000,A 180.000,B 0.000,C 180.000} C_DIS
LIN {X 122.587,Y 30.215,Z 52.000,A 180.000,B 0.000,C 180.000} C_DIS
LIN {X 122.850,Y 30.394,Z 52.000,A 180.000,B 0.000,C 180.000} C_DIS
LIN {X 122.997,Y 30.503,Z 52.000,A 180.000,B 0.000,C 180.000} C_DIS
LIN {X 123.176,Y 30.641,Z 52.000,A 180.000,B 0.000,C 180.000} C_DIS
LIN {X 123.313,Y 30.752,Z 52.000,A 180.000,B 0.000,C 180.000} C_DIS
LIN {X 123.533,Y 30.945,Z 52.000,A 180.000,B 0.000,C 180.000} C_DIS
LIN {X 123.709,Y 31.109,Z 52.000,A 180.000,B 0.000,C 180.000} C_DIS
LIN {X 123.891,Y 31.291,Z 52.000,A 180.000,B 0.000,C 180.000} C_DIS
LIN {X 124.055,Y 31.467,Z 52.000,A 180.000,B 0.000,C 180.000} C_DIS
LIN {X 124.248,Y 31.687,Z 52.000,A 180.000,B 0.000,C 180.000} C_DIS
LIN {X 124.359,Y 31.824,Z 52.000,A 180.000,B 0.000,C 180.000} C_DIS
LIN {X 124.497,Y 32.003,Z 52.000,A 180.000,B 0.000,C 180.000} C_DIS
LIN {X 124.606,Y 32.150,Z 52.000,A 180.000,B 0.000,C 180.000} C_DIS
LIN {X 124.785,Y 32.413,Z 52.000,A 180.000,B 0.000,C 180.000} C_DIS
LIN {X 124.865,Y 32.539,Z 52.000,A 180.000,B 0.000,C 180.000} C_DIS
LIN {X 124.971,Y 32.718,Z 52.000,A 180.000,B 0.000,C 180.000} C_DIS
LIN {X 125.076,Y 32.897,Z 52.000,A 180.000,B 0.000,C 180.000} C_DIS
LIN {X 125.258,Y 33.254,Z 52.000,A 180.000,B 0.000,C 180.000} C_DIS
LIN {X 125.321,Y 33.390,Z 52.000,A 180.000,B 0.000,C 180.000} C_DIS
LIN {X 125.417,Y 33.612,Z 52.000,A 180.000,B 0.000,C 180.000} C_DIS
LIN {X 125.491,Y 33.791,Z 52.000,A 180.000,B 0.000,C 180.000} C_DIS
LIN {X 125.619,Y 34.148,Z 52.000,A 180.000,B 0.000,C 180.000} C_DIS
LIN {X 125.674,Y 34.327,Z 52.000,A 180.000,B 0.000,C 180.000} C_DIS
LIN {X 125.726,Y 34.506,Z 52.000,A 180.000,B 0.000,C 180.000} C_DIS
LIN {X 125.774,Y 34.685,Z 52.000,A 180.000,B 0.000,C 180.000} C_DIS
LIN {X 125.857,Y 35.056,Z 52.000,A 180.000,B 0.000,C 180.000} C_DIS
LIN {X 125.886,Y 35.221,Z 52.000,A 180.000,B 0.000,C 180.000} C_DIS
LIN {X 125.914,Y 35.400,Z 52.000,A 180.000,B 0.000,C 180.000} C_DIS
LIN {X 125.941,Y 35.578,Z 52.000,A 180.000,B 0.000,C 180.000} C_DIS
LIN {X 125.975,Y 35.936,Z 52.000,A 180.000,B 0.000,C 180.000} C_DIS
LIN {X 125.987,Y 36.115,Z 52.000,A 180.000,B 0.000,C 180.000} C_DIS
LIN {X 125.998,Y 36.472,Z 52.000,A 180.000,B 0.000,C 180.000} C_DIS
LIN {X 125.994,Y 36.651,Z 52.000,A 180.000,B 0.000,C 180.000} C_DIS
LIN {X 125.988,Y 36.830,Z 52.000,A 180.000,B 0.000,C 180.000} C_DIS
LIN {X 125.980,Y 37.009,Z 52.000,A 180.000,B 0.000,C 180.000} C_DIS
LIN {X 125.947,Y 37.366,Z 52.000,A 180.000,B 0.000,C 180.000} C_DIS
LIN {X 125.923,Y 37.545,Z 52.000,A 180.000,B 0.000,C 180.000} C_DIS
LIN {X 125.866,Y 37.902,Z 52.000,A 180.000,B 0.000,C 180.000} C_DIS
LIN {X 125.857,Y 37.944,Z 52.000,A 180.000,B 0.000,C 180.000} C_DIS
LIN {X 125.787,Y 38.260,Z 52.000,A 180.000,B 0.000,C 180.000} C_DIS
LIN {X 125.742,Y 38.439,Z 52.000,A 180.000,B 0.000,C 180.000} C_DIS
LIN {X 125.638,Y 38.796,Z 52.000,A 180.000,B 0.000,C 180.000} C_DIS
LIN {X 125.575,Y 38.975,Z 52.000,A 180.000,B 0.000,C 180.000} C_DIS
LIN {X 125.500,Y 39.184,Z 52.000,A 180.000,B 0.000,C 180.000} C_DIS
LIN {X 125.441,Y 39.333,Z 52.000,A 180.000,B 0.000,C 180.000} C_DIS
LIN {X 125.286,Y 39.690,Z 52.000,A 180.000,B 0.000,C 180.000} C_DIS
LIN {X 125.195,Y 39.869,Z 52.000,A 180.000,B 0.000,C 180.000} C_DIS
LIN {X 125.104,Y 40.048,Z 52.000,A 180.000,B 0.000,C 180.000} C_DIS
LIN {X 125.004,Y 40.226,Z 52.000,A 180.000,B 0.000,C 180.000} C_DIS
LIN {X 124.898,Y 40.405,Z 52.000,A 180.000,B 0.000,C 180.000} C_DIS
LIN {X 124.787,Y 40.584,Z 52.000,A 180.000,B 0.000,C 180.000} C_DIS
LIN {X 124.606,Y 40.850,Z 52.000,A 180.000,B 0.000,C 180.000} C_DIS
LIN {X 124.540,Y 40.942,Z 52.000,A 180.000,B 0.000,C 180.000} C_DIS
LIN {X 124.402,Y 41.120,Z 52.000,A 180.000,B 0.000,C 180.000} C_DIS
LIN {X 124.261,Y 41.299,Z 52.000,A 180.000,B 0.000,C 180.000} C_DIS
LIN {X 124.070,Y 41.516,Z 52.000,A 180.000,B 0.000,C 180.000} C_DIS
LIN {X 123.943,Y 41.657,Z 52.000,A 180.000,B 0.000,C 180.000} C_DIS
LIN {X 123.712,Y 41.888,Z 52.000,A 180.000,B 0.000,C 180.000} C_DIS
LIN {X 123.579,Y 42.014,Z 52.000,A 180.000,B 0.000,C 180.000} C_DIS
LIN {X 123.354,Y 42.212,Z 52.000,A 180.000,B 0.000,C 180.000} C_DIS
LIN {X 123.176,Y 42.359,Z 52.000,A 180.000,B 0.000,C 180.000} C_DIS
LIN {X 122.928,Y 42.550,Z 52.000,A 180.000,B 0.000,C 180.000} C_DIS
LIN {X 122.818,Y 42.627,Z 52.000,A 180.000,B 0.000,C 180.000} C_DIS
LIN {X 122.639,Y 42.749,Z 52.000,A 180.000,B 0.000,C 180.000} C_DIS
LIN {X 122.461,Y 42.865,Z 52.000,A 180.000,B 0.000,C 180.000} C_DIS
LIN {X 122.282,Y 42.971,Z 52.000,A 180.000,B 0.000,C 180.000} C_DIS
LIN {X 122.103,Y 43.076,Z 52.000,A 180.000,B 0.000,C 180.000} C_DIS
LIN {X 121.731,Y 43.266,Z 52.000,A 180.000,B 0.000,C 180.000} C_DIS
LIN {X 121.567,Y 43.340,Z 52.000,A 180.000,B 0.000,C 180.000} C_DIS
LIN {X 121.325,Y 43.444,Z 52.000,A 180.000,B 0.000,C 180.000} C_DIS
LIN {X 121.209,Y 43.491,Z 52.000,A 180.000,B 0.000,C 180.000} C_DIS
LIN {X 120.841,Y 43.623,Z 52.000,A 180.000,B 0.000,C 180.000} C_DIS
LIN {X 120.673,Y 43.674,Z 52.000,A 180.000,B 0.000,C 180.000} C_DIS
LIN {X 120.494,Y 43.726,Z 52.000,A 180.000,B 0.000,C 180.000} C_DIS
LIN {X 120.315,Y 43.774,Z 52.000,A 180.000,B 0.000,C 180.000} C_DIS
LIN {X 119.958,Y 43.854,Z 52.000,A 180.000,B 0.000,C 180.000} C_DIS
LIN {X 119.779,Y 43.886,Z 52.000,A 180.000,B 0.000,C 180.000} C_DIS
LIN {X 119.600,Y 43.914,Z 52.000,A 180.000,B 0.000,C 180.000} C_DIS
LIN {X 119.422,Y 43.941,Z 52.000,A 180.000,B 0.000,C 180.000} C_DIS
LIN {X 119.006,Y 43.981,Z 52.000,A 180.000,B 0.000,C 180.000} C_DIS
LIN {X 118.885,Y 43.987,Z 52.000,A 180.000,B 0.000,C 180.000} C_DIS
LIN {X 118.528,Y 43.998,Z 52.000,A 180.000,B 0.000,C 180.000} C_DIS
LIN {X 118.349,Y 43.994,Z 52.000,A 180.000,B 0.000,C 180.000} C_DIS
LIN {X 118.170,Y 43.988,Z 52.000,A 180.000,B 0.000,C 180.000} C_DIS
LIN {X 117.994,Y 43.981,Z 52.000,A 180.000,B 0.000,C 180.000} C_DIS
LIN {X 117.634,Y 43.947,Z 52.000,A 180.000,B 0.000,C 180.000} C_DIS
LIN {X 117.455,Y 43.923,Z 52.000,A 180.000,B 0.000,C 180.000} C_DIS
LIN {X 117.098,Y 43.866,Z 52.000,A 180.000,B 0.000,C 180.000} C_DIS
LIN {X 116.919,Y 43.827,Z 52.000,A 180.000,B 0.000,C 180.000} C_DIS
LIN {X 116.740,Y 43.787,Z 52.000,A 180.000,B 0.000,C 180.000} C_DIS
LIN {X 116.561,Y 43.742,Z 52.000,A 180.000,B 0.000,C 180.000} C_DIS
LIN {X 116.204,Y 43.638,Z 52.000,A 180.000,B 0.000,C 180.000} C_DIS
LIN {X 116.159,Y 43.623,Z 52.000,A 180.000,B 0.000,C 180.000} C_DIS
LIN {X 115.846,Y 43.511,Z 52.000,A 180.000,B 0.000,C 180.000} C_DIS
LIN {X 115.675,Y 43.444,Z 52.000,A 180.000,B 0.000,C 180.000} C_DIS
LIN {X 115.310,Y 43.286,Z 52.000,A 180.000,B 0.000,C 180.000} C_DIS
LIN {X 115.269,Y 43.266,Z 52.000,A 180.000,B 0.000,C 180.000} C_DIS
LIN {X 114.918,Y 43.087,Z 52.000,A 180.000,B 0.000,C 180.000} C_DIS
LIN {X 114.774,Y 43.004,Z 52.000,A 180.000,B 0.000,C 180.000} C_DIS
LIN {X 114.595,Y 42.898,Z 52.000,A 180.000,B 0.000,C 180.000} C_DIS
LIN {X 114.416,Y 42.787,Z 52.000,A 180.000,B 0.000,C 180.000} C_DIS
LIN {X 114.237,Y 42.665,Z 52.000,A 180.000,B 0.000,C 180.000} C_DIS
LIN {X 114.072,Y 42.550,Z 52.000,A 180.000,B 0.000,C 180.000} C_DIS
LIN {X 113.841,Y 42.372,Z 52.000,A 180.000,B 0.000,C 180.000} C_DIS
LIN {X 113.701,Y 42.261,Z 52.000,A 180.000,B 0.000,C 180.000} C_DIS
LIN {X 113.421,Y 42.014,Z 52.000,A 180.000,B 0.000,C 180.000} C_DIS
LIN {X 113.343,Y 41.943,Z 52.000,A 180.000,B 0.000,C 180.000} C_DIS
LIN {X 113.057,Y 41.657,Z 52.000,A 180.000,B 0.000,C 180.000} C_DIS
LIN {X 112.986,Y 41.579,Z 52.000,A 180.000,B 0.000,C 180.000} C_DIS
LIN {X 112.739,Y 41.299,Z 52.000,A 180.000,B 0.000,C 180.000} C_DIS
LIN {X 112.628,Y 41.159,Z 52.000,A 180.000,B 0.000,C 180.000} C_DIS
LIN {X 112.450,Y 40.928,Z 52.000,A 180.000,B 0.000,C 180.000} C_DIS
LIN {X 112.335,Y 40.763,Z 52.000,A 180.000,B 0.000,C 180.000} C_DIS
LIN {X 112.213,Y 40.584,Z 52.000,A 180.000,B 0.000,C 180.000} C_DIS
LIN {X 112.102,Y 40.405,Z 52.000,A 180.000,B 0.000,C 180.000} C_DIS
LIN {X 111.996,Y 40.226,Z 52.000,A 180.000,B 0.000,C 180.000} C_DIS
LIN {X 111.913,Y 40.082,Z 52.000,A 180.000,B 0.000,C 180.000} C_DIS
LIN {X 111.734,Y 39.731,Z 52.000,A 180.000,B 0.000,C 180.000} C_DIS
LIN {X 111.714,Y 39.690,Z 52.000,A 180.000,B 0.000,C 180.000} C_DIS
LIN {X 111.556,Y 39.325,Z 52.000,A 180.000,B 0.000,C 180.000} C_DIS
LIN {X 111.489,Y 39.154,Z 52.000,A 180.000,B 0.000,C 180.000} C_DIS
LIN {X 111.377,Y 38.841,Z 52.000,A 180.000,B 0.000,C 180.000} C_DIS
LIN {X 111.362,Y 38.796,Z 52.000,A 180.000,B 0.000,C 180.000} C_DIS
LIN {X 111.258,Y 38.439,Z 52.000,A 180.000,B 0.000,C 180.000} C_DIS
LIN {X 111.213,Y 38.260,Z 52.000,A 180.000,B 0.000,C 180.000} C_DIS
LIN {X 111.173,Y 38.081,Z 52.000,A 180.000,B 0.000,C 180.000} C_DIS
LIN {X 111.134,Y 37.902,Z 52.000,A 180.000,B 0.000,C 180.000} C_DIS
LIN {X 111.077,Y 37.545,Z 52.000,A 180.000,B 0.000,C 180.000} C_DIS
LIN {X 111.053,Y 37.366,Z 52.000,A 180.000,B 0.000,C 180.000} C_DIS
LIN {X 111.019,Y 37.006,Z 52.000,A 180.000,B 0.000,C 180.000} C_DIS
LIN {X 111.012,Y 36.830,Z 52.000,A 180.000,B 0.000,C 180.000} C_DIS
LIN {X 111.006,Y 36.651,Z 52.000,A 180.000,B 0.000,C 180.000} C_DIS
LIN {X 111.002,Y 36.472,Z 52.000,A 180.000,B 0.000,C 180.000} C_DIS
LIN {X 111.013,Y 36.115,Z 52.000,A 180.000,B 0.000,C 180.000} C_DIS
LIN {X 111.019,Y 35.994,Z 52.000,A 180.000,B 0.000,C 180.000} C_DIS
LIN {X 111.059,Y 35.578,Z 52.000,A 180.000,B 0.000,C 180.000} C_DIS
LIN {X 111.086,Y 35.400,Z 52.000,A 180.000,B 0.000,C 180.000} C_DIS
LIN {X 111.114,Y 35.221,Z 52.000,A 180.000,B 0.000,C 180.000} C_DIS
LIN {X 111.146,Y 35.042,Z 52.000,A 180.000,B 0.000,C 180.000} C_DIS
LIN {X 111.226,Y 34.685,Z 52.000,A 180.000,B 0.000,C 180.000} C_DIS
LIN {X 111.274,Y 34.506,Z 52.000,A 180.000,B 0.000,C 180.000} C_DIS
LIN {X 111.326,Y 34.327,Z 52.000,A 180.000,B 0.000,C 180.000} C_DIS
LIN {X 111.377,Y 34.159,Z 52.000,A 180.000,B 0.000,C 180.000} C_DIS
LIN {X 111.509,Y 33.791,Z 52.000,A 180.000,B 0.000,C 180.000} C_DIS
LIN {X 111.556,Y 33.675,Z 52.000,A 180.000,B 0.000,C 180.000} C_DIS
LIN {X 111.660,Y 33.433,Z 52.000,A 180.000,B 0.000,C 180.000} C_DIS
LIN {X 111.734,Y 33.269,Z 52.000,A 180.000,B 0.000,C 180.000} C_DIS
LIN {X 111.924,Y 32.897,Z 52.000,A 180.000,B 0.000,C 180.000} C_DIS
LIN {X 112.029,Y 32.718,Z 52.000,A 180.000,B 0.000,C 180.000} C_DIS
LIN {X 112.121,Y 32.562,Z 52.000,A 180.000,B 0.000,C 180.000} C_DIS
; Lead Out Move Starts
LIN {X 112.511,Y 32.318,Z 52.000,A 180.000,B 0.000,C 180.000} C_DIS
LIN {X 112.935,Y 32.496,Z 52.000,A 180.000,B 0.000,C 180.000} C_DIS
LIN {X 113.522,Y 33.197,Z 52.000,A 180.000,B 0.000,C 180.000} C_DIS
LIN {X 113.749,Y 33.468,Z 52.146,A 180.000,B 0.000,C 180.000} C_DIS
LIN {X 113.844,Y 33.580,Z 52.500,A 180.000,B 0.000,C 180.000} C_DIS
; Rapid Move Starts
LIN {X 113.844,Y 33.580,Z 95.000,A 180.000,B 0.000,C 180.000} C_DIS
LIN {X 42.599,Y 35.562,Z 95.000,A 180.000,B 0.000,C 180.000} C_DIS
LIN {X 42.599,Y 35.562,Z 58.499,A 180.000,B 0.000,C 180.000} C_DIS
; Plunge Move Starts
$VEL.CP=0.01
LIN {X 42.599,Y 35.562,Z 57.625,A 180.000,B 0.000,C 180.000} C_DIS
; Lead In Move Starts
LIN {X 42.599,Y 35.562,Z 56.500,A 180.000,B 0.000,C 180.000} C_DIS
LIN {X 42.745,Y 35.555,Z 56.146,A 180.000,B 0.000,C 180.000} C_DIS
LIN {X 43.099,Y 35.537,Z 56.000,A 180.000,B 0.000,C 180.000} C_DIS
LIN {X 43.456,Y 35.519,Z 56.000,A 180.000,B 0.000,C 180.000} C_DIS
LIN {X 43.817,Y 35.648,Z 56.000,A 180.000,B 0.000,C 180.000} C_DIS
LIN {X 43.981,Y 35.994,Z 56.000,A 180.000,B 0.000,C 180.000} C_DIS
; Cutting Move Starts
$VEL.CP=0.02
LIN {X 43.987,Y 36.115,Z 56.000,A 180.000,B 0.000,C 180.000} C_DIS
LIN {X 43.998,Y 36.472,Z 56.000,A 180.000,B 0.000,C 180.000} C_DIS
LIN {X 43.994,Y 36.651,Z 56.000,A 180.000,B 0.000,C 180.000} C_DIS
LIN {X 43.988,Y 36.830,Z 56.000,A 180.000,B 0.000,C 180.000} C_DIS
LIN {X 43.981,Y 37.006,Z 56.000,A 180.000,B 0.000,C 180.000} C_DIS
LIN {X 43.947,Y 37.366,Z 56.000,A 180.000,B 0.000,C 180.000} C_DIS
LIN {X 43.923,Y 37.545,Z 56.000,A 180.000,B 0.000,C 180.000} C_DIS
LIN {X 43.866,Y 37.902,Z 56.000,A 180.000,B 0.000,C 180.000} C_DIS
LIN {X 43.827,Y 38.081,Z 56.000,A 180.000,B 0.000,C 180.000} C_DIS
LIN {X 43.787,Y 38.260,Z 56.000,A 180.000,B 0.000,C 180.000} C_DIS
LIN {X 43.742,Y 38.439,Z 56.000,A 180.000,B 0.000,C 180.000} C_DIS
LIN {X 43.638,Y 38.796,Z 56.000,A 180.000,B 0.000,C 180.000} C_DIS
LIN {X 43.623,Y 38.841,Z 56.000,A 180.000,B 0.000,C 180.000} C_DIS
LIN {X 43.511,Y 39.154,Z 56.000,A 180.000,B 0.000,C 180.000} C_DIS
LIN {X 43.444,Y 39.325,Z 56.000,A 180.000,B 0.000,C 180.000} C_DIS
LIN {X 43.286,Y 39.690,Z 56.000,A 180.000,B 0.000,C 180.000} C_DIS
LIN {X 43.266,Y 39.731,Z 56.000,A 180.000,B 0.000,C 180.000} C_DIS
LIN {X 43.087,Y 40.082,Z 56.000,A 180.000,B 0.000,C 180.000} C_DIS
LIN {X 43.004,Y 40.226,Z 56.000,A 180.000,B 0.000,C 180.000} C_DIS
LIN {X 42.898,Y 40.405,Z 56.000,A 180.000,B 0.000,C 180.000} C_DIS
LIN {X 42.787,Y 40.584,Z 56.000,A 180.000,B 0.000,C 180.000} C_DIS
LIN {X 42.665,Y 40.763,Z 56.000,A 180.000,B 0.000,C 180.000} C_DIS
LIN {X 42.550,Y 40.928,Z 56.000,A 180.000,B 0.000,C 180.000} C_DIS
LIN {X 42.372,Y 41.159,Z 56.000,A 180.000,B 0.000,C 180.000} C_DIS
LIN {X 42.261,Y 41.299,Z 56.000,A 180.000,B 0.000,C 180.000} C_DIS
LIN {X 42.014,Y 41.579,Z 56.000,A 180.000,B 0.000,C 180.000} C_DIS
LIN {X 41.943,Y 41.657,Z 56.000,A 180.000,B 0.000,C 180.000} C_DIS
LIN {X 41.657,Y 41.943,Z 56.000,A 180.000,B 0.000,C 180.000} C_DIS
LIN {X 41.579,Y 42.014,Z 56.000,A 180.000,B 0.000,C 180.000} C_DIS
LIN {X 41.299,Y 42.261,Z 56.000,A 180.000,B 0.000,C 180.000} C_DIS
LIN {X 41.159,Y 42.372,Z 56.000,A 180.000,B 0.000,C 180.000} C_DIS
LIN {X 40.928,Y 42.550,Z 56.000,A 180.000,B 0.000,C 180.000} C_DIS
LIN {X 40.763,Y 42.665,Z 56.000,A 180.000,B 0.000,C 180.000} C_DIS
LIN {X 40.584,Y 42.787,Z 56.000,A 180.000,B 0.000,C 180.000} C_DIS
LIN {X 40.405,Y 42.898,Z 56.000,A 180.000,B 0.000,C 180.000} C_DIS
LIN {X 40.226,Y 43.004,Z 56.000,A 180.000,B 0.000,C 180.000} C_DIS
LIN {X 40.082,Y 43.087,Z 56.000,A 180.000,B 0.000,C 180.000} C_DIS
LIN {X 39.731,Y 43.266,Z 56.000,A 180.000,B 0.000,C 180.000} C_DIS
LIN {X 39.690,Y 43.286,Z 56.000,A 180.000,B 0.000,C 180.000} C_DIS
LIN {X 39.325,Y 43.444,Z 56.000,A 180.000,B 0.000,C 180.000} C_DIS
LIN {X 39.154,Y 43.511,Z 56.000,A 180.000,B 0.000,C 180.000} C_DIS
LIN {X 38.841,Y 43.623,Z 56.000,A 180.000,B 0.000,C 180.000} C_DIS
LIN {X 38.796,Y 43.638,Z 56.000,A 180.000,B 0.000,C 180.000} C_DIS
LIN {X 38.439,Y 43.742,Z 56.000,A 180.000,B 0.000,C 180.000} C_DIS
LIN {X 38.260,Y 43.787,Z 56.000,A 180.000,B 0.000,C 180.000} C_DIS
LIN {X 38.081,Y 43.827,Z 56.000,A 180.000,B 0.000,C 180.000} C_DIS
LIN {X 37.902,Y 43.866,Z 56.000,A 180.000,B 0.000,C 180.000} C_DIS
LIN {X 37.545,Y 43.923,Z 56.000,A 180.000,B 0.000,C 180.000} C_DIS
LIN {X 37.366,Y 43.947,Z 56.000,A 180.000,B 0.000,C 180.000} C_DIS
LIN {X 37.006,Y 43.981,Z 56.000,A 180.000,B 0.000,C 180.000} C_DIS
LIN {X 36.830,Y 43.988,Z 56.000,A 180.000,B 0.000,C 180.000} C_DIS
LIN {X 36.651,Y 43.994,Z 56.000,A 180.000,B 0.000,C 180.000} C_DIS
LIN {X 36.472,Y 43.998,Z 56.000,A 180.000,B 0.000,C 180.000} C_DIS
LIN {X 36.115,Y 43.987,Z 56.000,A 180.000,B 0.000,C 180.000} C_DIS
LIN {X 35.994,Y 43.981,Z 56.000,A 180.000,B 0.000,C 180.000} C_DIS
LIN {X 35.578,Y 43.941,Z 56.000,A 180.000,B 0.000,C 180.000} C_DIS
LIN {X 35.400,Y 43.914,Z 56.000,A 180.000,B 0.000,C 180.000} C_DIS
LIN {X 35.221,Y 43.886,Z 56.000,A 180.000,B 0.000,C 180.000} C_DIS
LIN {X 35.042,Y 43.854,Z 56.000,A 180.000,B 0.000,C 180.000} C_DIS
LIN {X 34.685,Y 43.774,Z 56.000,A 180.000,B 0.000,C 180.000} C_DIS
LIN {X 34.506,Y 43.726,Z 56.000,A 180.000,B 0.000,C 180.000} C_DIS
LIN {X 34.327,Y 43.674,Z 56.000,A 180.000,B 0.000,C 180.000} C_DIS
LIN {X 34.159,Y 43.623,Z 56.000,A 180.000,B 0.000,C 180.000} C_DIS
LIN {X 33.791,Y 43.491,Z 56.000,A 180.000,B 0.000,C 180.000} C_DIS
LIN {X 33.675,Y 43.444,Z 56.000,A 180.000,B 0.000,C 180.000} C_DIS
LIN {X 33.433,Y 43.340,Z 56.000,A 180.000,B 0.000,C 180.000} C_DIS
LIN {X 33.269,Y 43.266,Z 56.000,A 180.000,B 0.000,C 180.000} C_DIS
LIN {X 32.897,Y 43.076,Z 56.000,A 180.000,B 0.000,C 180.000} C_DIS
LIN {X 32.718,Y 42.971,Z 56.000,A 180.000,B 0.000,C 180.000} C_DIS
LIN {X 32.539,Y 42.865,Z 56.000,A 180.000,B 0.000,C 180.000} C_DIS
LIN {X 32.361,Y 42.749,Z 56.000,A 180.000,B 0.000,C 180.000} C_DIS
LIN {X 32.182,Y 42.627,Z 56.000,A 180.000,B 0.000,C 180.000} C_DIS
LIN {X 32.072,Y 42.550,Z 56.000,A 180.000,B 0.000,C 180.000} C_DIS
LIN {X 31.824,Y 42.359,Z 56.000,A 180.000,B 0.000,C 180.000} C_DIS
LIN {X 31.646,Y 42.212,Z 56.000,A 180.000,B 0.000,C 180.000} C_DIS
LIN {X 31.421,Y 42.014,Z 56.000,A 180.000,B 0.000,C 180.000} C_DIS
LIN {X 31.288,Y 41.888,Z 56.000,A 180.000,B 0.000,C 180.000} C_DIS
LIN {X 31.057,Y 41.657,Z 56.000,A 180.000,B 0.000,C 180.000} C_DIS
LIN {X 30.930,Y 41.516,Z 56.000,A 180.000,B 0.000,C 180.000} C_DIS
LIN {X 30.739,Y 41.299,Z 56.000,A 180.000,B 0.000,C 180.000} C_DIS
LIN {X 30.598,Y 41.120,Z 56.000,A 180.000,B 0.000,C 180.000} C_DIS
LIN {X 30.460,Y 40.942,Z 56.000,A 180.000,B 0.000,C 180.000} C_DIS
LIN {X 30.394,Y 40.850,Z 56.000,A 180.000,B 0.000,C 180.000} C_DIS
LIN {X 30.213,Y 40.584,Z 56.000,A 180.000,B 0.000,C 180.000} C_DIS
LIN {X 30.102,Y 40.405,Z 56.000,A 180.000,B 0.000,C 180.000} C_DIS
LIN {X 29.996,Y 40.226,Z 56.000,A 180.000,B 0.000,C 180.000} C_DIS
LIN {X 29.896,Y 40.048,Z 56.000,A 180.000,B 0.000,C 180.000} C_DIS
LIN {X 29.805,Y 39.869,Z 56.000,A 180.000,B 0.000,C 180.000} C_DIS
LIN {X 29.714,Y 39.690,Z 56.000,A 180.000,B 0.000,C 180.000} C_DIS
LIN {X 29.559,Y 39.333,Z 56.000,A 180.000,B 0.000,C 180.000} C_DIS
LIN {X 29.500,Y 39.184,Z 56.000,A 180.000,B 0.000,C 180.000} C_DIS
LIN {X 29.425,Y 38.975,Z 56.000,A 180.000,B 0.000,C 180.000} C_DIS
LIN {X 29.362,Y 38.796,Z 56.000,A 180.000,B 0.000,C 180.000} C_DIS
LIN {X 29.258,Y 38.439,Z 56.000,A 180.000,B 0.000,C 180.000} C_DIS
LIN {X 29.213,Y 38.260,Z 56.000,A 180.000,B 0.000,C 180.000} C_DIS
LIN {X 29.143,Y 37.944,Z 56.000,A 180.000,B 0.000,C 180.000} C_DIS
LIN {X 29.134,Y 37.902,Z 56.000,A 180.000,B 0.000,C 180.000} C_DIS
LIN {X 29.077,Y 37.545,Z 56.000,A 180.000,B 0.000,C 180.000} C_DIS
LIN {X 29.053,Y 37.366,Z 56.000,A 180.000,B 0.000,C 180.000} C_DIS
LIN {X 29.020,Y 37.009,Z 56.000,A 180.000,B 0.000,C 180.000} C_DIS
LIN {X 29.012,Y 36.830,Z 56.000,A 180.000,B 0.000,C 180.000} C_DIS
LIN {X 29.006,Y 36.651,Z 56.000,A 180.000,B 0.000,C 180.000} C_DIS
LIN {X 29.002,Y 36.472,Z 56.000,A 180.000,B 0.000,C 180.000} C_DIS
LIN {X 29.013,Y 36.115,Z 56.000,A 180.000,B 0.000,C 180.000} C_DIS
LIN {X 29.025,Y 35.936,Z 56.000,A 180.000,B 0.000,C 180.000} C_DIS
LIN {X 29.059,Y 35.578,Z 56.000,A 180.000,B 0.000,C 180.000} C_DIS
LIN {X 29.086,Y 35.400,Z 56.000,A 180.000,B 0.000,C 180.000} C_DIS
LIN {X 29.114,Y 35.221,Z 56.000,A 180.000,B 0.000,C 180.000} C_DIS
LIN {X 29.143,Y 35.056,Z 56.000,A 180.000,B 0.000,C 180.000} C_DIS
LIN {X 29.226,Y 34.685,Z 56.000,A 180.000,B 0.000,C 180.000} C_DIS
LIN {X 29.274,Y 34.506,Z 56.000,A 180.000,B 0.000,C 180.000} C_DIS
LIN {X 29.326,Y 34.327,Z 56.000,A 180.000,B 0.000,C 180.000} C_DIS
LIN {X 29.381,Y 34.148,Z 56.000,A 180.000,B 0.000,C 180.000} C_DIS
LIN {X 29.509,Y 33.791,Z 56.000,A 180.000,B 0.000,C 180.000} C_DIS
LIN {X 29.583,Y 33.612,Z 56.000,A 180.000,B 0.000,C 180.000} C_DIS
LIN {X 29.679,Y 33.390,Z 56.000,A 180.000,B 0.000,C 180.000} C_DIS
LIN {X 29.742,Y 33.254,Z 56.000,A 180.000,B 0.000,C 180.000} C_DIS
LIN {X 29.924,Y 32.897,Z 56.000,A 180.000,B 0.000,C 180.000} C_DIS
LIN {X 30.029,Y 32.718,Z 56.000,A 180.000,B 0.000,C 180.000} C_DIS
LIN {X 30.135,Y 32.539,Z 56.000,A 180.000,B 0.000,C 180.000} C_DIS
LIN {X 30.215,Y 32.413,Z 56.000,A 180.000,B 0.000,C 180.000} C_DIS
LIN {X 30.394,Y 32.150,Z 56.000,A 180.000,B 0.000,C 180.000} C_DIS
LIN {X 30.503,Y 32.003,Z 56.000,A 180.000,B 0.000,C 180.000} C_DIS
LIN {X 30.641,Y 31.824,Z 56.000,A 180.000,B 0.000,C 180.000} C_DIS
LIN {X 30.752,Y 31.687,Z 56.000,A 180.000,B 0.000,C 180.000} C_DIS
LIN {X 30.945,Y 31.467,Z 56.000,A 180.000,B 0.000,C 180.000} C_DIS
LIN {X 31.109,Y 31.291,Z 56.000,A 180.000,B 0.000,C 180.000} C_DIS
LIN {X 31.291,Y 31.109,Z 56.000,A 180.000,B 0.000,C 180.000} C_DIS
LIN {X 31.467,Y 30.945,Z 56.000,A 180.000,B 0.000,C 180.000} C_DIS
LIN {X 31.687,Y 30.752,Z 56.000,A 180.000,B 0.000,C 180.000} C_DIS
LIN {X 31.824,Y 30.641,Z 56.000,A 180.000,B 0.000,C 180.000} C_DIS
LIN {X 32.003,Y 30.503,Z 56.000,A 180.000,B 0.000,C 180.000} C_DIS
LIN {X 32.150,Y 30.394,Z 56.000,A 180.000,B 0.000,C 180.000} C_DIS
LIN {X 32.413,Y 30.215,Z 56.000,A 180.000,B 0.000,C 180.000} C_DIS
LIN {X 32.539,Y 30.135,Z 56.000,A 180.000,B 0.000,C 180.000} C_DIS
LIN {X 32.718,Y 30.029,Z 56.000,A 180.000,B 0.000,C 180.000} C_DIS
LIN {X 32.897,Y 29.924,Z 56.000,A 180.000,B 0.000,C 180.000} C_DIS
LIN {X 33.254,Y 29.742,Z 56.000,A 180.000,B 0.000,C 180.000} C_DIS
LIN {X 33.390,Y 29.679,Z 56.000,A 180.000,B 0.000,C 180.000} C_DIS
LIN {X 33.612,Y 29.583,Z 56.000,A 180.000,B 0.000,C 180.000} C_DIS
LIN {X 33.791,Y 29.509,Z 56.000,A 180.000,B 0.000,C 180.000} C_DIS
LIN {X 34.148,Y 29.381,Z 56.000,A 180.000,B 0.000,C 180.000} C_DIS
LIN {X 34.327,Y 29.326,Z 56.000,A 180.000,B 0.000,C 180.000} C_DIS
LIN {X 34.506,Y 29.274,Z 56.000,A 180.000,B 0.000,C 180.000} C_DIS
LIN {X 34.685,Y 29.226,Z 56.000,A 180.000,B 0.000,C 180.000} C_DIS
LIN {X 35.056,Y 29.143,Z 56.000,A 180.000,B 0.000,C 180.000} C_DIS
LIN {X 35.221,Y 29.114,Z 56.000,A 180.000,B 0.000,C 180.000} C_DIS
LIN {X 35.400,Y 29.086,Z 56.000,A 180.000,B 0.000,C 180.000} C_DIS
LIN {X 35.578,Y 29.059,Z 56.000,A 180.000,B 0.000,C 180.000} C_DIS
LIN {X 35.936,Y 29.025,Z 56.000,A 180.000,B 0.000,C 180.000} C_DIS
LIN {X 36.115,Y 29.013,Z 56.000,A 180.000,B 0.000,C 180.000} C_DIS
LIN {X 36.472,Y 29.002,Z 56.000,A 180.000,B 0.000,C 180.000} C_DIS
LIN {X 36.651,Y 29.006,Z 56.000,A 180.000,B 0.000,C 180.000} C_DIS
LIN {X 36.830,Y 29.012,Z 56.000,A 180.000,B 0.000,C 180.000} C_DIS
LIN {X 37.009,Y 29.020,Z 56.000,A 180.000,B 0.000,C 180.000} C_DIS
LIN {X 37.366,Y 29.053,Z 56.000,A 180.000,B 0.000,C 180.000} C_DIS
LIN {X 37.545,Y 29.077,Z 56.000,A 180.000,B 0.000,C 180.000} C_DIS
LIN {X 37.902,Y 29.134,Z 56.000,A 180.000,B 0.000,C 180.000} C_DIS
LIN {X 37.944,Y 29.143,Z 56.000,A 180.000,B 0.000,C 180.000} C_DIS
LIN {X 38.260,Y 29.213,Z 56.000,A 180.000,B 0.000,C 180.000} C_DIS
LIN {X 38.439,Y 29.258,Z 56.000,A 180.000,B 0.000,C 180.000} C_DIS
LIN {X 38.796,Y 29.362,Z 56.000,A 180.000,B 0.000,C 180.000} C_DIS
LIN {X 38.975,Y 29.425,Z 56.000,A 180.000,B 0.000,C 180.000} C_DIS
LIN {X 39.184,Y 29.500,Z 56.000,A 180.000,B 0.000,C 180.000} C_DIS
LIN {X 39.333,Y 29.559,Z 56.000,A 180.000,B 0.000,C 180.000} C_DIS
LIN {X 39.690,Y 29.714,Z 56.000,A 180.000,B 0.000,C 180.000} C_DIS
LIN {X 39.869,Y 29.805,Z 56.000,A 180.000,B 0.000,C 180.000} C_DIS
LIN {X 40.048,Y 29.896,Z 56.000,A 180.000,B 0.000,C 180.000} C_DIS
LIN {X 40.226,Y 29.996,Z 56.000,A 180.000,B 0.000,C 180.000} C_DIS
LIN {X 40.405,Y 30.102,Z 56.000,A 180.000,B 0.000,C 180.000} C_DIS
LIN {X 40.584,Y 30.213,Z 56.000,A 180.000,B 0.000,C 180.000} C_DIS
LIN {X 40.850,Y 30.394,Z 56.000,A 180.000,B 0.000,C 180.000} C_DIS
LIN {X 40.942,Y 30.460,Z 56.000,A 180.000,B 0.000,C 180.000} C_DIS
LIN {X 41.120,Y 30.598,Z 56.000,A 180.000,B 0.000,C 180.000} C_DIS
LIN {X 41.299,Y 30.739,Z 56.000,A 180.000,B 0.000,C 180.000} C_DIS
LIN {X 41.516,Y 30.930,Z 56.000,A 180.000,B 0.000,C 180.000} C_DIS
LIN {X 41.657,Y 31.057,Z 56.000,A 180.000,B 0.000,C 180.000} C_DIS
LIN {X 41.888,Y 31.288,Z 56.000,A 180.000,B 0.000,C 180.000} C_DIS
LIN {X 42.014,Y 31.421,Z 56.000,A 180.000,B 0.000,C 180.000} C_DIS
LIN {X 42.212,Y 31.646,Z 56.000,A 180.000,B 0.000,C 180.000} C_DIS
LIN {X 42.359,Y 31.824,Z 56.000,A 180.000,B 0.000,C 180.000} C_DIS
LIN {X 42.550,Y 32.072,Z 56.000,A 180.000,B 0.000,C 180.000} C_DIS
LIN {X 42.627,Y 32.182,Z 56.000,A 180.000,B 0.000,C 180.000} C_DIS
LIN {X 42.749,Y 32.361,Z 56.000,A 180.000,B 0.000,C 180.000} C_DIS
LIN {X 42.865,Y 32.539,Z 56.000,A 180.000,B 0.000,C 180.000} C_DIS
LIN {X 42.971,Y 32.718,Z 56.000,A 180.000,B 0.000,C 180.000} C_DIS
LIN {X 43.076,Y 32.897,Z 56.000,A 180.000,B 0.000,C 180.000} C_DIS
LIN {X 43.266,Y 33.269,Z 56.000,A 180.000,B 0.000,C 180.000} C_DIS
LIN {X 43.340,Y 33.433,Z 56.000,A 180.000,B 0.000,C 180.000} C_DIS
LIN {X 43.444,Y 33.675,Z 56.000,A 180.000,B 0.000,C 180.000} C_DIS
LIN {X 43.491,Y 33.791,Z 56.000,A 180.000,B 0.000,C 180.000} C_DIS
LIN {X 43.623,Y 34.159,Z 56.000,A 180.000,B 0.000,C 180.000} C_DIS
LIN {X 43.674,Y 34.327,Z 56.000,A 180.000,B 0.000,C 180.000} C_DIS
LIN {X 43.726,Y 34.506,Z 56.000,A 180.000,B 0.000,C 180.000} C_DIS
LIN {X 43.774,Y 34.685,Z 56.000,A 180.000,B 0.000,C 180.000} C_DIS
LIN {X 43.854,Y 35.042,Z 56.000,A 180.000,B 0.000,C 180.000} C_DIS
LIN {X 43.886,Y 35.221,Z 56.000,A 180.000,B 0.000,C 180.000} C_DIS
LIN {X 43.914,Y 35.400,Z 56.000,A 180.000,B 0.000,C 180.000} C_DIS
LIN {X 43.941,Y 35.578,Z 56.000,A 180.000,B 0.000,C 180.000} C_DIS
LIN {X 43.981,Y 35.994,Z 56.000,A 180.000,B 0.000,C 180.000} C_DIS
; Link Move Starts
LIN {X 43.993,Y 36.309,Z 56.000,A 180.000,B 0.000,C 180.000} C_DIS
LIN {X 43.995,Y 36.624,Z 55.999,A 180.000,B 0.000,C 180.000} C_DIS
LIN {X 43.985,Y 36.938,Z 55.998,A 180.000,B 0.000,C 180.000} C_DIS
